// SIMATIC S7-200 SMART project (STEP 7-Micro/WIN SMART), CPU ST20

SYMBOL_TABLE 系统符号
Always_On        SM0.0    // 始终接通
First_Scan_On    SM0.1    // 仅在第一个扫描周期时接通
Clock_60s        SM0.4    // 针对 1 分钟的周期时间，时钟脉冲接通 30 s，断开 30 s.
Clock_1s         SM0.5    // 针对 1 s 的周期时间，时钟脉冲接通 0.5 s，断开 0.5 s.
END_SYMBOL_TABLE

ORGANIZATION_BLOCK MAIN:OB1
TITLE=// ============================================================
// // 文件: OB1_MAIN.stl
// // 功能: PLC主循环程序
// // 项目: 药液配置与加注控制系统
// // Story: AQEX-6 状态机骨架 + AQEX-9 急停调度顺序确认
// // PLC: S7-200 SMART CPU ST20
// // 说明: 本文件为语句表(STL)格式，可参考导入STEP 7-Micro/WIN SMART
// // 调度顺序: FC0(初始化)→FC2(急停,最高优先级)→FC4(Modbus)→FC3(报警)→FC22(RTC同步)
// //           →FC40(双倒计时器周期管理,v2.2新增)→FC1(状态调度)
// //           FC2在FC1之前,保证急停触发时同周期转S_ERROR
// //           FC40在FC1之前,保证M16.1下一轮S1触发脉冲及时响应
// //           【v2.2 修订 2026-09-15】FC40 从 FC1 内部调用移至 OB1 顶层调度
// // ============================================================
// 
// // 符号注释（实际导入时在符号表定义）
// // VW2     : 状态机当前状态 (0=S0,1=S1...8=S7,99=ERROR)
// // VW4     : 注射泵状态码
// // VW6     : 当前最高优先级报警码
// // VW8     : 实验总换水次数目标(=VD414×VD24/1440,单位:次)
// // V0.0    : CMD_Start (HMI→PLC启动命令)
// // V0.2    : CMD_Stop  (HMI→PLC停止命令)
// // V1.0    : STA_StartAck (PLC→HMI启动确认)
// // I1.1    : DI_EStop (急停反馈，常开NO，OFF=正常/ON=急停触发)  v1.3 改NO接法(原"常闭,ON=正常"注释已过期)
// // I0.3    : DI_Btn_SystemReset (系统复位按钮)
// 
BEGIN
Network 1
//  首次扫描初始化
//  SM0.1仅在首次扫描周期ON，调用FC0系统初始化
LD     First_Scan_On:SM0.1
=      L60.0                 // 局部存储器中转
LD     L60.0
CALL   SysInit:SBR0




// 急停与安全处理（每周期调用，优先级最高）
     // 急停与安全处理（每周期调用，优先级最高）
// SM0.0常ON，每周期调用FC2
        // SM0.0常ON，每周期调用FC2
LD     Always_On:SM0.0
CALL   EStopHandling:SBR2




// HMI停止命令(V0.2) - 自动运行中任意状态可停止
 // HMI停止命令(V0.2) - 自动运行中任意状态可停止
// ★ 2026-09-11 修复:
         // ★ 2026-09-11 修复:
//   (1) 去掉 AW< VW2, 99 条件,允许 S_ERROR 态(VW2=99)也能停止
 //   (1) 去掉 AW< VW2, 99 条件,允许 S_ERROR 态(VW2=99)也能停止
//       原逻辑只允许 VW2=1~8 停止, S_ERROR 锁死时点停止被忽略
 //       原逻辑只允许 VW2=1~8 停止, S_ERROR 锁死时点停止被忽略
//       新逻辑: VW2>0(非S0)就能停止, 急停/继电器故障锁存位由 FC19 管理
 //       新逻辑: VW2>0(非S0)就能停止, 急停/继电器故障锁存位由 FC19 管理
//   (2) 补清阀门诊断子状态 VB260~VB275 和诊断计时器 T50~T55
 //   (2) 补清阀门诊断子状态 VB260~VB275 和诊断计时器 T50~T55
//       原三个清理路径(停止/冷启动/复位)全部遗漏,导致
 //       原三个清理路径(停止/冷启动/复位)全部遗漏,导致
//       FC11/FC15/FC17 的 AW=VW2xx,0 前置条件不成立,
 //       FC11/FC15/FC17 的 AW=VW2xx,0 前置条件不成立,
//       开阀指令被跳过,表现为"点启动 M10.2=1 但系统不运行"
 //       开阀指令被跳过,表现为"点启动 M10.2=1 但系统不运行"
LD     V0.2
EU
AW>    VW2, 0                // VW2>0(排除S0), VW2=1~8 或 99 都允许停止
LPS
R      CPU_输出0:Q0.0, 7       // 泵停/阀关/NC电磁阀失电
R      T37, 1                // 停S1计时器
R      M10.2, 1              // 清S1首次进入标志
R      M10.7, 1              // 清预规划标志
R      M11.6, 1              // 清注射泵写请求
// ★ 新增: 清阀门诊断子状态+结果(VB260~VB275, 8字=16字节)
 // ★ 新增: 清阀门诊断子状态+结果(VB260~VB275, 8字=16字节)
//   覆盖: 阀A子状态VB260~261, 阀B子状态VB262~263,
 //   覆盖: 阀A子状态VB260~261, 阀B子状态VB262~263,
//         阀A/B结果VB266~269, 阀C诊断VB270~273, 其他辅助变量
 //         阀A/B结果VB266~269, 阀C诊断VB270~273, 其他辅助变量
FILL   0, VW260, 8
// ★ 新增: 清阀A/B诊断计时器 T50~T55
 // ★ 新增: 清阀A/B诊断计时器 T50~T55
R      T50, 6
// 【v2.2新增】停止时清理上缸子流程状态 + 双倒计时器标志 + 定时器
 // 【v2.2新增】停止时清理上缸子流程状态 + 双倒计时器标志 + 定时器
MOVW   0, VW418              // 上缸配液子流程状态清零
MOVW   0, VW400              // 换水计数清零 【v2.3.2迁移: 原VW306与手动命令位V306.0~V307.3重叠】
R      M16.0, 4              // M16.0~M16.3 连续清零
R      T38, 1                // 清 S2 搅拌定时器
R      T63, 1                // [已修复 v2.2] 清 1s 脉冲定时器
R      T49, 1                // 清 S4 转移计时器
MOVR   0.0, VD248            // [已修复 v2.2] 清 TimerA_Elapsed
MOVR   0.0, VD252            // [已修复 v2.2] 清 TimerB_Elapsed
MOVR   0.0, VD256            // 清 TimerA 显示值
MOVR   0.0, VD244            // 清 TimerB 显示值
MOVW   0, VW2                // 回S0
R      V0.2, 1               // 清停止命令
LPP




// Modbus通讯轮询（每周期调用）
        // Modbus通讯轮询（每周期调用）
LD     Always_On:SM0.0
CALL   ModbusPolling:SBR4




// 报警处理（每周期调用）
              // 报警处理（每周期调用）
LD     Always_On:SM0.0
CALL   AlarmHandling:SBR3




// RTC时间同步处理（每周期调用）
         // RTC时间同步处理（每周期调用）
// 处理HMI校时命令V0.6和5分钟超时保护
    // 处理HMI校时命令V0.6和5分钟超时保护
LD     Always_On:SM0.0
CALL   RTC_Sync:SBR24




// v2.2 双倒计时器周期管理（每周期调用）
    // v2.2 双倒计时器周期管理（每周期调用）
// ★ 必须在 FC1 状态调度之前调用,保证 M16.1 下一轮 S1 触发脉冲及时响应
 // ★ 必须在 FC1 状态调度之前调用,保证 M16.1 下一轮 S1 触发脉冲及时响应
// 替代原 AQEX-8 三层纠偏,严格保证 24h 换水次数硬约束 (VD414)
 // 替代原 AQEX-8 三层纠偏,严格保证 24h 换水次数硬约束 (VD414)
// 功能: 计算 T_cycle / 触发 S6 / 触发下一轮 S1 / 倒计时到 0 报警 / 双计时器显示值
 // 功能: 计算 T_cycle / 触发 S6 / 触发下一轮 S1 / 倒计时到 0 报警 / 双计时器显示值
LD     Always_On:SM0.0
CALL   RhythmCorrection:SBR19




// 【v2.3 新增】M16.1 唯一消费点: FC40 触发下一轮 S1 → 上缸 VW418 4→1
 // 【v2.3 新增】M16.1 唯一消费点: FC40 触发下一轮 S1 → 上缸 VW418 4→1
// 置位方只有 FC40 NET5 (Prep_Needed 且距周期末 ≥ T_prep), FC10/FC15 不再置位
 // 置位方只有 FC40 NET5 (Prep_Needed 且距周期末 ≥ T_prep), FC10/FC15 不再置位
// 【2026-09-29修复】同步置 M10.2(S1首次进入标志),与FC10首轮播种口径一致,
 // 【2026-09-29修复】同步置 M10.2(S1首次进入标志),与FC10首轮播种口径一致,
//   否则下一轮S1因FC11入口门(LD M10.2)不通而空转
 //   否则下一轮S1因FC11入口门(LD M10.2)不通而空转
LD     M16.1
MOVW   1, VW418
S      M10.2, 1
R      M16.1, 1




// 状态机调度(急停时FC2会强制VW2=99)
   // 状态机调度(急停时FC2会强制VW2=99)
// 每周期根据VW2调用对应状态FC
         // 每周期根据VW2调用对应状态FC
LD     Always_On:SM0.0
CALL   StateDispatcher:SBR1




// 【v2.2 新增】上缸子流程调度(VW418)
  // 【v2.2 新增】上缸子流程调度(VW418)
// 在 FC1 下缸调度之后调用,处理上缸 S1/S2 并行流程
 // 在 FC1 下缸调度之后调用,处理上缸 S1/S2 并行流程
// VW418=1 → CALL FC11_State_S1_Inlet (上缸进水)
 // VW418=1 → CALL FC11_State_S1_Inlet (上缸进水)
// VW418=2 → CALL FC1A_State_S2_MixDose (上缸搅拌+加药合并,v2.2 新建)
 // VW418=2 → CALL FC1A_State_S2_MixDose (上缸搅拌+加药合并,v2.2 新建)
// VW418=0/3/4 → 无动作(空闲/配完等待/已转移由其他 FC 处理)
 // VW418=0/3/4 → 无动作(空闲/配完等待/已转移由其他 FC 处理)
LD     Always_On:SM0.0
AW=    VW418, 1
AW>    VW2, 0                // 【2026-09-24修复】非S0(上缸随下缸运行才允许执行)
AW<    VW2, 99               // 【2026-09-24修复】非S_ERROR(故障锁定禁止上缸动作)
CALL   State_S1_Inlet:SBR6
LD     Always_On:SM0.0
AW=    VW418, 2
AW>    VW2, 0                // 【2026-09-24修复】同上
AW<    VW2, 99               // 【2026-09-24修复】同上
CALL   State_S2_MixDose:SBR7




// 手动控制处理（仅在S0态调用,在状态调度之后）
  // 手动控制处理（仅在S0态调用,在状态调度之后）
// 处理HMI画面3手动控制命令位V306.0~V307.1
 // 处理HMI画面3手动控制命令位V306.0~V307.1
//   (旧地址V2.4~V3.5因与VW2物理重叠已于2026-09-03迁移,详见FC20符号表)
 //   (旧地址V2.4~V3.5因与VW2物理重叠已于2026-09-03迁移,详见FC20符号表)
// 由FC20使用M13.0~M13.4锁存输出,NC电磁阀自动跟随(详见FC20)
 // 由FC20使用M13.0~M13.4锁存输出,NC电磁阀自动跟随(详见FC20)
LD     Always_On:SM0.0
LDW=   VW2, 0
CALL   ManualControl:SBR15




// 手动注射泵控制（仅在S0态调用,在手动阀门控制之后）
 // 手动注射泵控制（仅在S0态调用,在手动阀门控制之后）
// 处理V307.2/V307.3命令位
       // 处理V307.2/V307.3命令位
//   (旧地址V3.6/V3.7因与VW2物理重叠已于2026-09-03迁移,详见FC21符号表)
 //   (旧地址V3.6/V3.7因与VW2物理重叠已于2026-09-03迁移,详见FC21符号表)
// 【v2.5】由FC21壳使用VD452/VW388/VW390执行单次/循环抽排,
 // 【v2.5】由FC21壳使用VD452/VW388/VW390执行单次/循环抽排,
//   泵协议状态机与自动共用FC23引擎(详见FC21/FC23)
 //   泵协议状态机与自动共用FC23引擎(详见FC21/FC23)
LD     Always_On:SM0.0
LDW=   VW2, 0
CALL   ManualSyringePump:SBR23




// 非S0态清除手动控制锁存与手动注射泵状态,防止返回S0时误动作
 // 非S0态清除手动控制锁存与手动注射泵状态,防止返回S0时误动作
// 【v2.5】M13.5/M13.6保护标志已退役(FC23引擎取消),只清停止请求M13.7;
 // 【v2.5】M13.5/M13.6保护标志已退役(FC23引擎取消),只清停止请求M13.7;
//   追加手动模式残留子状态清除: 自动运行期间FC13壳已把M17.0刷0条件恒假,
 //   追加手动模式残留子状态清除: 自动运行期间FC13壳已把M17.0刷0条件恒假,
//   手动中途切自动时M17.0=1→清VW226,防引擎带旧子状态进入自动路径
 //   手动中途切自动时M17.0=1→清VW226,防引擎带旧子状态进入自动路径
LD     Always_On:SM0.0
LDW=   VW2, 0
NOT
R      M13.0, 5              // 清阀门/泵手动锁存
R      M13.7, 1              // 清停止请求(v2.5: M13.5/13.6已退役)
MOVW   0, VW390              // HMI状态镜像复位(空闲)
LDW=   VW2, 0
NOT
A      M17.0                 // 【v2.5】VW2≠0 且 手动模式残留
MOVW   0, VW226              // 清引擎子状态(FC23与FC13/FC21共用)
R      M17.0, 1




// M16.4/5/6 → V区镜像（供HMI读取，McgsPro S7-200 SMART以太网驱动不支持M区直接导入）
 // M16.4/5/6 → V区镜像（供HMI读取，McgsPro S7-200 SMART以太网驱动不支持M区直接导入）
// V1.1=InitDone(原M16.4), V1.2=RTU1/Syringe在线(原M16.5), V0.1=RTU2/Flow在线(原M16.6)
 // V1.1=InitDone(原M16.4), V1.2=RTU1/Syringe在线(原M16.5), V0.1=RTU2/Flow在线(原M16.6)
LD     Always_On:SM0.0
LD     M16.4
=      V1.1
LD     M16.5
=      V1.2
LD     M16.6
=      V0.1




// 系统总状态 → VB305 (0=良好,1=故障,2=急停)
 // 系统总状态 → VB305 (0=良好,1=故障,2=急停)
// 急停: I1.1=ON(NO触点,ON=急停触发) OR V300.4 OR V300.5
 // 急停: I1.1=ON(NO触点,ON=急停触发) OR V300.4 OR V300.5
// 故障: VW6≠0 AND 非急停
        // 故障: VW6≠0 AND 非急停
// 良好: 非急停 AND VW6=0 (默认值)
  // 良好: 非急停 AND VW6=0 (默认值)
// 【2026-09-24修复】v1.3改NO接法后此处漏改: 原"LD I1.1 / NOT"把I1.1=OFF(正常)误判为急停,
 // 【2026-09-24修复】v1.3改NO接法后此处漏改: 原"LD I1.1 / NOT"把I1.1=OFF(正常)误判为急停,
//   导致急停释放后HMI标题栏永久显示"急停"; 故障分支的"A I1.1"同步改为"AN I1.1"
 //   导致急停释放后HMI标题栏永久显示"急停"; 故障分支的"A I1.1"同步改为"AN I1.1"


LD     Always_On:SM0.0
MOVB   0, VB305              // 默认良好
// 急停 → 2
                   // 急停 → 2
LD     CPU_输入9:I1.1          // NO触点: ON=急停触发
O      V300.4
O      V300.5
MOVB   2, VB305
// 非急停 + 有报警 → 1
            // 非急停 + 有报警 → 1
LDW<>  VW6, 0
AN     CPU_输入9:I1.1          // 急停未触发(NO触点OFF=正常)
AN     V300.4
AN     V300.5
MOVB   1, VB305




// 实验总换水次数目标计算(v2.2新增)
      // 实验总换水次数目标计算(v2.2新增)
// VW8 = VD414(24h换水目标次数) × VD24(实验总时长min) / 1440
 // VW8 = VD414(24h换水目标次数) × VD24(实验总时长min) / 1440
// 供HMI画面显示实验全程应完成的总换水次数
    // 供HMI画面显示实验全程应完成的总换水次数
LD     Always_On:SM0.0
MOVR   VD414, AC0
*R     VD24, AC0
/R     1440.0, AC0
ROUND  AC0, AC0
DTI    AC0, VW8




// ============================================================
 // ============================================================
// 文件结束
                     // 文件结束
// 说明:
                      // 说明:
//   1. FC0/FC1/FC2/FC3/FC4 见各自独立文件
 //   1. FC0/FC1/FC2/FC3/FC4 见各自独立文件
//   2. FC10~FC19 各状态FC见 State_Sxx.stl 文件
 //   2. FC10~FC19 各状态FC见 State_Sxx.stl 文件
//   3. FC20 手动控制(新增,AQEX-34修复)
 //   3. FC20 手动控制(新增,AQEX-34修复)
//   4. FC22 RTC时间同步处理(新增,AQEX-51)
 //   4. FC22 RTC时间同步处理(新增,AQEX-51)
//   5. 导入时需先建符号表，再逐个新建FC并粘贴代码
 //   5. 导入时需先建符号表，再逐个新建FC并粘贴代码
//   6. VB305 系统状态字(=0良好/1故障/2急停,AQEX-50新增)
 //   6. VB305 系统状态字(=0良好/1故障/2急停,AQEX-50新增)
// ============================================================
 // ============================================================


END_ORGANIZATION_BLOCK

SUBROUTINE_BLOCK SysInit:SBR0
TITLE=// ============================================================
// // 文件: FC0_SysInit.stl (调度骨架)
// // 功能: 系统初始化入口 — 首次扫描 + Modbus清零 + 冷启/断电路径调度
// // Story: AQEX-6 + AQEX-11 + AQEX-51
// // 说明: 拆分自原单一 FC0,冷启/断电恢复逻辑分别独立到 SBR25/SBR26
// //   跨 SBR 无 JMP/LBL 依赖,每个 SBR 内部 LBL 空间独立
// // LBL 分配: FC0 用 1(断电恢复入口)、2(完成汇合)
// //          SBR25 用 8/9/10/88/89(冷启动)
// //          SBR26 用 1/3/4/5/6/7(断电恢复)
// //   跨 SBR 编号相同不冲突,POU 内 LBL 空间独立
// // 修复记录:
// //   2026-09-13: 拆分前 FC0 12KB 导致 STEP7 下载"块过大"误判,
// //               拆分后 FC0(~3KB) + SBR25(~4KB) + SBR26(~4KB) 三个小块
// // ============================================================
// 
// // 符号说明:
// // M16.4: M_InitDone        初始化完成标志(断电保持;v2.2迁移自V304.0,2026-09-15)
// // VW198 : VW_Init_Step      初始化步骤号(调试用,0=完成)
// // ColdStart  : SBR25 冷启动路径
// // WarmRecovery: SBR26 断电恢复路径
// 
// 
BEGIN
Network 1
//  SM0.1首次扫描 + Modbus库清零 + FC21计数器清零
//  ★ 2026-09-07修复: 每次首次扫描统一清零,库状态机在STOP→RUN后必须复位
LD     First_Scan_On:SM0.1
MOVW   1, VW198


LD     First_Scan_On:SM0.1
FILL   0, VW600, 143         // VB600~VB885清零(Modbus库存储区)
FILL   0, VW378, 2           // 清 VB378~VB381 (MBUS Error 4字节合并)
R      M10.0, 6              // 清M10.0~M10.5(Done位/降级标志)
R      M11.0, 1              // 清MBUS_CTRL Done位
MOVW   0, VW390              // 清手动注射泵子状态
R      M11.6, 1              // 清注射泵写请求
R      T104, 1               // 清回零冷却定时器




// 冷启/断电路径调度 + 完成汇合
         // 冷启/断电路径调度 + 完成汇合
// 判断冷启动/断电恢复
               // 判断冷启动/断电恢复
// M16.4=1 → JMP 1 (LBL 1: CALL WarmRecovery → JMP 2)
 // M16.4=1 → JMP 1 (LBL 1: CALL WarmRecovery → JMP 2)
// M16.4=0 → 冷启动 → CALL ColdStart → RET回 FC0 继续到 LBL 2
 // M16.4=0 → 冷启动 → CALL ColdStart → RET回 FC0 继续到 LBL 2
// 【v2.2迁移 2026-09-15】M_InitDone 从 V304.0 迁至 M16.4（位对象，无字节级冲突）
 // 【v2.2迁移 2026-09-15】M_InitDone 从 V304.0 迁至 M16.4（位对象，无字节级冲突）


LD     M16.4
JMP    1                     // M16.4=1 → 跳断电恢复路径


// ========== 冷启动路径 ==========
 // ========== 冷启动路径 ==========
LD     First_Scan_On:SM0.1
AN     M16.4                 // 冷启动(M16.4=0)
CALL   ColdStart:SBR25       // SBR25: 出厂硬编码 + 用户默认覆盖 + TODR + 安全初始化
                          // ColdStart 自然结束返回
 // ColdStart 自然结束返回
LD     Always_On:SM0.0
JMP    2                     // ★ 关键: 无条件跳过 LBL 1,否则会形成死循环


// ========== 断电恢复路径 ==========
 // ========== 断电恢复路径 ==========
LBL    1
LD     First_Scan_On:SM0.1
CALL   WarmRecovery:SBR26    // SBR26: TODR + RTC检测 + BCD转秒 + 状态机恢复
                          // WarmRecovery 自然结束后,顺序执行到 LBL 2 汇合
 // WarmRecovery 自然结束后,顺序执行到 LBL 2 汇合


// ========== 初始化完成汇合 ==========
 // ========== 初始化完成汇合 ==========
LBL    2
LD     First_Scan_On:SM0.1
S      M16.4, 1              // M_InitDone=1(初始化完成,断电保持;从V304.0迁移)
MOVW   0, VW198              // 步骤=0(完成)
// 汇合后自然结束 FC0,返回 OB1
       // 汇合后自然结束 FC0,返回 OB1




// ============================================================
 // ============================================================
// 文件结束
                     // 文件结束
// ============================================================
 // ============================================================


END_SUBROUTINE_BLOCK

SUBROUTINE_BLOCK StateDispatcher:SBR1
TITLE=// ============================================================
// // 文件: FC1_StateDispatcher.stl
// // 功能: 状态机调度器（每周期根据VW2调用对应下缸状态FC）
// // Story: v2.2 流程重构 (替代 AQEX-6 状态机骨架)
// // 说明: v2.2 取消上缸流程作为下缸主状态的 S1/S2/S3/S3.5
// //       上缸流程已拆出到 VW418 State_UpTank 子流程,由 OB1 NET 7 直接调度
// //       本 FC1 仅调度下缸 VW2 路径: S0/S4/S5/S6/S7/S_ERROR
// //   修复记录:
// //     P1-NETWORK标题去掉冒号(错误66)
// //     P2-JMP/LBL跨NETWORK问题修复: 全部合并到NETWORK 1
// //     【v2.2 修订 2026-09-15】删除 S1/S2/S3/S3.5 LBL;上缸流程外移至 OB1
// // ============================================================
BEGIN
Network 1
//  状态调度 (JMP/LBL必须在同一NETWORK内)
//  读取VW2并与各状态值比较，相等则调用对应FC
//  VW2 = 0 → S0初始化
JMP    1
// VW2 = 5 → S4上→下转移         // VW2 = 5 → S4上→下转移
LDW=   VW2, 5
JMP    2
// VW2 = 6 → S5实验运行中         // VW2 = 6 → S5实验运行中
LDW=   VW2, 6
JMP    3
// VW2 = 7 → S6下缸排水          // VW2 = 7 → S6下缸排水
LDW=   VW2, 7
JMP    4
// VW2 = 8 → S7实验结束          // VW2 = 8 → S7实验结束
LDW=   VW2, 8
JMP    5
// VW2 = 99 → S_ERROR故障锁定    // VW2 = 99 → S_ERROR故障锁定
LDW=   VW2, 99
JMP    6
// 其他非法值 → 强制回S0             // 其他非法值 → 强制回S0
LDW>=  VW2, 100
JMP    7
// 若未匹配任何状态(0<VW2<99但非上述值),也回S0 // 若未匹配任何状态(0<VW2<99但非上述值),也回S0
JMP    7
// S0入口                      // S0入口
LBL    1
CALL State_S0_Init
JMP    8
// S4入口                      // S4入口
LBL    2
CALL State_S4_Transfer
JMP    8
// S5入口                      // S5入口
LBL    3
CALL State_S5_Run
JMP    8
// S6入口                      // S6入口
LBL    4
CALL State_S6_Drain
JMP    8
// S7入口                      // S7入口
LBL    5
CALL State_S7_End
JMP    8
// S_ERROR入口                 // S_ERROR入口
LBL    6
CALL State_Error
JMP    8
// 非法状态处理(强制回S0)             // 非法状态处理(强制回S0)
LBL    7
LDW<=  VW2, 0                // VW2=0
// 调度结束                      // 调度结束
LBL    8
// 状态调度完成,返回 OB1             // 状态调度完成,返回 OB1
// 注: 上缸子流程(VW418=1/2)由 OB1 NET 7 在本 FC1 之后调度 // 注: 上缸子流程(VW418=1/2)由 OB1 NET 7 在本 FC1 之后调度
// ============================================================ // ============================================================
// 文件结束                      // 文件结束
// 说明:                       // 说明:
//   1. JMP/LBL必须在同一NETWORK内 //   1. JMP/LBL必须在同一NETWORK内
//   2. 每个状态FC内部负责状态转移(修改VW2) //   2. 每个状态FC内部负责状态转移(修改VW2)
//   3. 【v2.2】删除 S1/S2/S3/S3.5 入口:上缸流程移至 VW418 子流程 //   3. 【v2.2】删除 S1/S2/S3/S3.5 入口:上缸流程移至 VW418 子流程
//   4. 【v2.2】VW2 路径:0(S0)→5(S4)→6(S5)→7(S6)→8(S7) 或 99(S_ERROR) //   4. 【v2.2】VW2 路径:0(S0)→5(S4)→6(S5)→7(S6)→8(S7) 或 99(S_ERROR)
//   5. 【v2.2】VW418 路径:0(空闲)→1(S1)→2(S2搅拌+加药)→4(已转移) //   5. 【v2.2】VW418 路径:0(空闲)→1(S1)→2(S2搅拌+加药)→4(已转移)
//                          或 3(配完等待),由 OB1 NET 7 调度 FC11/FC1A //                          或 3(配完等待),由 OB1 NET 7 调度 FC11/FC1A
// ============================================================
 // ============================================================
JMP    1
LDW=   VW2, 5
JMP    2
LDW=   VW2, 6
JMP    3
LDW=   VW2, 7
JMP    4
LDW=   VW2, 8
JMP    5
LDW=   VW2, 99
JMP    6
LDW>=  VW2, 100
JMP    7
JMP    7
LBL    1
CALL   State_S0_Init:SBR5
JMP    8
LBL    2
CALL   State_S4_Transfer:SBR10
JMP    8
LBL    3
CALL   State_S5_Run:SBR11
JMP    8
LBL    4
CALL   State_S6_Drain:SBR12
JMP    8
LBL    5
CALL   State_S7_End:SBR13
JMP    8
LBL    6
CALL   State_Error:SBR14
JMP    8
LBL    7
MOVW   0, VW2
LBL    8
END_SUBROUTINE_BLOCK

SUBROUTINE_BLOCK EStopHandling:SBR2
TITLE=// ============================================================
// // 文件: FC2_EStopHandling.stl
// // 功能: 急停与安全处理（每周期调用，优先级最高）
// // Story: AQEX-6 状态机骨架 + AQEX-9 急停双通道+安全继电器反馈(详细实现)
// // 说明: 急停检测(I1.1 上升沿:NO 闭合)→锁存V300.4→转S_ERROR  v1.3 NO 进 I1.1
// //       安全继电器反馈延时校验(2秒)→V300.5继电器故障最高级报警
// //       输出强制安全(QB0=0,Q0.7声音开)
// //       急停解除与系统复位由FC19(State_Error)处理
// // ============================================================
// 
// // 符号说明:
// // I1.1  : DI_EStop           急停反馈(常开 NO,OFF=正常,ON=急停触发)  v1.3 改为接 NO 触点
// // I1.2  : DI_SafetyRelay_FB  安全继电器辅助反馈(ON=动力回路接通,OFF=动力回路断开)
// // V300.4: M_EStop_Latch      急停触发锁存(漫溢级,强制人工确认)
// // V300.5: M_Alarm_SafetyRelay 安全继电器故障(最高级,强制人工确认)
// // VW2   : 状态机状态(FC2写99转S_ERROR)
// // VW6   : 报警码(99=继电器故障,10=急停)
// // T35   : 安全继电器反馈延时(PT=20,2秒)
// // M10.7 : 预规划触发标志(急停时清,防止S5残留)
// 
// 
BEGIN
Network 1
//  急停触发+锁存+转S_ERROR + 安全继电器反馈校验 + 输出强制安全(合并NET 1-3)
//  [已修复 v2.2] 用 V62.6 缓存 EU 结果,避免 S/R 链栈空;删除直接写 VW6(由 FC3 根据 V300.x 计算)
LD     CPU_输入9:I1.1
EU
AN     First_Scan_On:SM0.1   // 首次扫描周期不触发（调试临时）
=      V62.6
LD     V62.6
S      V300.4, 1             // M_EStop_Latch锁存
LD     V62.6
MOVW   99, VW2               // VW2=99(转S_ERROR)
LD     V62.6
R      M10.7, 1              // 清预规划标志


// 安全继电器反馈延时校验(2秒内I1.2应OFF,否则继电器故障)
 // 安全继电器反馈延时校验(2秒内I1.2应OFF,否则继电器故障)
LD     V300.4
A      CPU_输入10:I1.2
TON    T35, 20
LD     T35
EU
S      V300.5, 1             // M_Alarm_SafetyRelay


// 急停锁存时输出强制安全
              // 急停锁存时输出强制安全
LD     V300.4
MOVB   0, QB0                // 泵停/阀关/NC电磁阀失电(安全)
S      CPU_输出7:Q0.7, 1       // 报警声音开




// 报警码写入(优先级:继电器故障99 > 急停10)
 // 报警码写入(优先级:继电器故障99 > 急停10)
// [已修复 v2.2] 删除直接写 VW6,统一由 FC3 NETWORK1 根据 V300.4/V300.5 计算
 // [已修复 v2.2] 删除直接写 VW6,统一由 FC3 NETWORK1 根据 V300.4/V300.5 计算
// LD     V300.5
            // LD     V300.5
// MOVW   99, VW6
           // MOVW   99, VW6
// LD     V300.4
            // LD     V300.4
// AN     V300.5
            // AN     V300.5
// MOVW   10, VW6
           // MOVW   10, VW6


LBL    1




// 注: HMI停止命令由OB1 MAIN NETWORK 3统一处理(VW2>0即可停止),本FC不再处理
 // 注: HMI停止命令由OB1 MAIN NETWORK 3统一处理(VW2>0即可停止),本FC不再处理
// 注: 急停解除与系统复位逻辑在FC19(State_Error)中处理
 // 注: 急停解除与系统复位逻辑在FC19(State_Error)中处理
// 注: Q8.0报警灯光由FC3 AlarmHandling按VW6优先级统一管理(Story 1.6)
 // 注: Q8.0报警灯光由FC3 AlarmHandling按VW6优先级统一管理(Story 1.6)
// 注: I1.2接线逻辑:ON=动力回路接通,OFF=动力回路断开(与代码注释一致)
 // 注: I1.2接线逻辑:ON=动力回路接通,OFF=动力回路断开(与代码注释一致)
// 注: 安全继电器反馈延时2秒兼顾机械动作时间与故障捕获灵敏度
 // 注: 安全继电器反馈延时2秒兼顾机械动作时间与故障捕获灵敏度
// 注: 急停硬件回路(安全继电器切断动力电)不经过PLC,本FC仅处理软件层面
 // 注: 急停硬件回路(安全继电器切断动力电)不经过PLC,本FC仅处理软件层面




// ============================================================
 // ============================================================
// 文件结束
                     // 文件结束
// ============================================================
 // ============================================================


END_SUBROUTINE_BLOCK

SUBROUTINE_BLOCK AlarmHandling:SBR3
TITLE=// ============================================================
// // 文件: FC3_AlarmHandling.stl
// // 功能: 报警处理（每周期调用）
// // Story: AQEX-6 状态机骨架 + AQEX-10 报警分级与消音/消光逻辑(详细实现)
// // 说明: 优先级链计算VW6 + 消音(I0.4/V0.4) + 消光(V0.3确认)
// //       自动恢复模式(V200.0=0时一般故障级条件消失自动复位)
// //       高优先级(漫溢/节奏滞后/继电器故障)强制人工确认,不受模式影响
// // ============================================================
// 
// // 符号说明:
// // VW6   : 当前最高优先级未确认报警码(0=无,99=继电器故障,10~14漫溢,20~21节奏,30~65一般)
// // V200.0: M_AlarmAckMode 报警确认模式(0=自动恢复,1=人工确认)
// // Q0.7  : 报警声音(FC2/FC19置位,FC3管理消音)
// // Q8.0  : 报警灯光(FC3统一管理,避免双写冲突)
// // I0.4  : 就地消音按钮(常开点动)
// // V0.3  : CMD_AckAlarm HMI报警确认命令
// // V0.4  : CMD_Mute HMI消音命令
// // V1.3  : STA_AlarmAckDone 报警确认握手
// // V1.4  : STA_MuteDone 消音握手
// // M11.1 : M_Sound_Latched 声音已消音标志(新报警时清,实现重鸣)
// // M11.2 : M_PrevAlarm 上一周期有报警标志(新报警检测用)
// 
// 
BEGIN
Network 1
//  优先级链计算 VW6(最高优先级未确认报警码)
//  压缩版: 用 LDW=+A+MOVW 条件赋值,替代 LD/JMP/LBL 结构
//  优先级: 99 > 10~14 > 20~21 > 66 > 30~36 > 40~47 > 49 > 60~61 > 64~65
//  【v10.4硬件变更】链中已移除: 13(V300.3)/45(V302.5)/47(V302.7)/61(V303.1),
//    对应位均改为保留位,当前有效码不含13/45/47/61
//  原理: 从最高优先级开始逐个检查,VW6一旦被赋值,后续 LDW= VW6,0 为假,自动跳过
LD     Always_On:SM0.0
MOVW   0, VW6                // 默认无报警


// 1. 安全继电器故障(99)
           // 1. 安全继电器故障(99)
LD     V300.5
MOVW   99, VW6


// 2. 漫溢级(10~14) - 逐位检查
     // 2. 漫溢级(10~14) - 逐位检查
// 【v10.4硬件变更】报警码13(V300.3,原NC球阀-下缸动作)已废弃,
 // 【v10.4硬件变更】报警码13(V300.3,原NC球阀-下缸动作)已废弃,
//   Q0.6去除后无任何FC置位V300.3,优先级链移除该条目(V300.3为保留位)
 //   Q0.6去除后无任何FC置位V300.3,优先级链移除该条目(V300.3为保留位)
LDW=   VW6, 0
A      V300.0
MOVW   10, VW6
LDW=   VW6, 0
A      V300.1
MOVW   11, VW6
LDW=   VW6, 0
A      V300.2
MOVW   12, VW6
LDW=   VW6, 0
A      V300.4
MOVW   14, VW6


// 3. 节奏滞后(20~21)
           // 3. 节奏滞后(20~21)
LDW=   VW6, 0
A      V300.6
MOVW   20, VW6
LDW=   VW6, 0
A      V300.7
MOVW   21, VW6


// 4. 单轮换水周期超时(66)
          // 4. 单轮换水周期超时(66)
LDW=   VW6, 0
A      V303.6
MOVW   66, VW6


// 5. 阀A类(30~36) - 逐位检查
     // 5. 阀A类(30~36) - 逐位检查
LDW=   VW6, 0
A      V301.0
MOVW   30, VW6
LDW=   VW6, 0
A      V301.2
MOVW   32, VW6
LDW=   VW6, 0
A      V301.3
MOVW   33, VW6
LDW=   VW6, 0
A      V301.4
MOVW   34, VW6
LDW=   VW6, 0
A      V301.5
MOVW   35, VW6
LDW=   VW6, 0
A      V301.6
MOVW   36, VW6


// 6. 阀B/C类(40~47) - 逐位检查
   // 6. 阀B/C类(40~47) - 逐位检查
// 【v10.4硬件变更】报警码45(V302.5)/47(V302.7)已废弃(I0.2去除,FC32不再置位),
 // 【v10.4硬件变更】报警码45(V302.5)/47(V302.7)已废弃(I0.2去除,FC32不再置位),
//   优先级链移除该两条目(V302.5/V302.7为保留位)
 //   优先级链移除该两条目(V302.5/V302.7为保留位)
LDW=   VW6, 0
A      V302.0
MOVW   40, VW6
LDW=   VW6, 0
A      V302.1
MOVW   41, VW6
LDW=   VW6, 0
A      V302.2
MOVW   42, VW6
LDW=   VW6, 0
A      V302.3
MOVW   43, VW6
LDW=   VW6, 0
A      V302.4
MOVW   44, VW6
LDW=   VW6, 0
A      V302.6
MOVW   46, VW6


// 7. 其他类(49,60,64,65)
      // 7. 其他类(49,60,64,65)
// 【v10.4硬件变更】报警码61(V303.1,原阀C关到位仍有流)已废弃(内漏判定依赖I0.2),
 // 【v10.4硬件变更】报警码61(V303.1,原阀C关到位仍有流)已废弃(内漏判定依赖I0.2),
//   优先级链移除该条目;报警码60(V303.0)现覆盖关到位超时+排水超时两种触发
 //   优先级链移除该条目;报警码60(V303.0)现覆盖关到位超时+排水超时两种触发
LDW=   VW6, 0
A      V303.2
MOVW   49, VW6
LDW=   VW6, 0
A      V303.0
MOVW   60, VW6
LDW=   VW6, 0
A      V303.4
MOVW   64, VW6
LDW=   VW6, 0
A      V303.5
MOVW   65, VW6




// 报警输出管理(灯光常亮 + 新报警声音重鸣)
   // 报警输出管理(灯光常亮 + 新报警声音重鸣)
// 有活动报警(VW6≠0) → 灯光Q8.0常亮
  // 有活动报警(VW6≠0) → 灯光Q8.0常亮
// 新报警(VW6由0变非0) → 清M_Sound_Latched,声音重鸣
 // 新报警(VW6由0变非0) → 清M_Sound_Latched,声音重鸣
LDW<>  VW6, 0
S      EM0_输出0:Q8.0, 1       // 灯光常亮


// 新报警检测: 本周期VW6≠0 且 上一周期M11.2=0(无报警) → 新报警
 // 新报警检测: 本周期VW6≠0 且 上一周期M11.2=0(无报警) → 新报警
LDW<>  VW6, 0
AN     M11.2                 // 上一周期无报警 → 新报警
R      M11.1, 1              // 清消音标志(新报警重鸣)


// 声音管理: 有报警且未消音 → 声音开
      // 声音管理: 有报警且未消音 → 声音开
LDW<>  VW6, 0
AN     M11.1                 // 未消音
S      CPU_输出7:Q0.7, 1       // 声音开


// 自动恢复模式: VW6=0且自动模式 → 自动消光
 // 自动恢复模式: VW6=0且自动模式 → 自动消光
LDW=   VW6, 0
AN     V200.0                // M_AlarmAckMode=0(自动模式)
R      EM0_输出0:Q8.0, 1       // 无报警自动消光
R      CPU_输出7:Q0.7, 1       // 无报警关声音
R      M11.1, 1              // 清消音标志


// 更新上一周期报警标志
               // 更新上一周期报警标志
LDW<>  VW6, 0
=      M11.2                 // 记录本周期有报警(供下周期新报警检测)




// 消音处理(I0.4就地按钮 OR V0.4 HMI命令)
 // 消音处理(I0.4就地按钮 OR V0.4 HMI命令)
// [已修复 v2.2] 用 V62.7 缓存消音请求,避免 OLD 后 S/R 链栈空
 // [已修复 v2.2] 用 V62.7 缓存消音请求,避免 OLD 后 S/R 链栈空
// 消音源: I0.4上升沿 OR V0.4上升沿
  // 消音源: I0.4上升沿 OR V0.4上升沿
LD     CPU_输入4:I0.4
EU
LD     V0.4
EU
OLD                          // 两者任一上升沿
=      V62.7
LD     V62.7
R      CPU_输出7:Q0.7, 1       // 关声音
LD     V62.7
S      M11.1, 1              // 置消音标志(新报警时清)
LD     V62.7
S      V1.4, 1               // STA_MuteDone握手
LD     V62.7
R      V0.4, 1               // 清HMI消音命令
// 注: 消音只关声音,灯光Q8.0和报警位保持;新报警(VW6变化)时M11.1清,声音重鸣
 // 注: 消音只关声音,灯光Q8.0和报警位保持;新报警(VW6变化)时M11.1清,声音重鸣




// 报警确认处理(V0.3 HMI确认 → 条件消失才消光+清锁存)
 // 报警确认处理(V0.3 HMI确认 → 条件消失才消光+清锁存)
// V0.3上升沿 = HMI报警确认命令(高优先级HMI侧二次确认,PLC只收V0.3)
 // V0.3上升沿 = HMI报警确认命令(高优先级HMI侧二次确认,PLC只收V0.3)
// 确认规则: V0.3上升沿后,逐个检查报警位条件,条件消失的复位报警位,再由NETWORK1重算VW6
 // 确认规则: V0.3上升沿后,逐个检查报警位条件,条件消失的复位报警位,再由NETWORK1重算VW6
// ★ 关键修复(2026-09-04): NETWORK 4 缺 V0.3 上升沿门控(JMP),导致每周期无条件
 // ★ 关键修复(2026-09-04): NETWORK 4 缺 V0.3 上升沿门控(JMP),导致每周期无条件
//   执行所有条件复位,包括 LD V303.5; R V303.5, 1——使 S_ERROR 立即被清
 //   执行所有条件复位,包括 LD V303.5; R V303.5, 1——使 S_ERROR 立即被清
//   修复: V0.3 无上升沿时跳过整个网络,避免误清报警位
 //   修复: V0.3 无上升沿时跳过整个网络,避免误清报警位
// ★★★ 2026-09-11 发现 JMP 条件写反了！ ★★★
 // ★★★ 2026-09-11 发现 JMP 条件写反了！ ★★★
//   原代码 LD V0.3; EU; JMP 40：EU=1(有上升沿)时跳转 → 反而跳过了 R V0.3,1
 //   原代码 LD V0.3; EU; JMP 40：EU=1(有上升沿)时跳转 → 反而跳过了 R V0.3,1
//   正确：用 V60.5 缓存 EU 结果,LDN 取反后触发 JMP,再用 LD 恢复栈顶执行线圈
 //   正确：用 V60.5 缓存 EU 结果,LDN 取反后触发 JMP,再用 LD 恢复栈顶执行线圈
//   注意：STL 的 S/R/= 线圈指令依赖栈顶=1 才执行,不能用 NOT+JMP（会清掉栈顶）
 //   注意：STL 的 S/R/= 线圈指令依赖栈顶=1 才执行,不能用 NOT+JMP（会清掉栈顶）
//   注意：S7-200 SMART 不支持 JMPN 指令,必须用 JMP + LDN 中转
 //   注意：S7-200 SMART 不支持 JMPN 指令,必须用 JMP + LDN 中转
LD     V0.3
EU
=      V60.5                 // 缓存 EU 结果: 有上升沿=1, 无上升沿=0
LDN    V60.5                 // 无上升沿时栈顶=1
JMP    40                    // ★ 无上升沿则跳转到 LBL 40,跳过确认处理
LD     V60.5                 // 有上升沿时栈顶=1,恢复执行条件


S      V1.3, 1               // STA_AlarmAckDone握手
R      V0.3, 1               // 清确认命令


// 漫溢级: 条件消失才复位(液位计高位=OFF)
  // 漫溢级: 条件消失才复位(液位计高位=OFF)
LD     V300.0                // 上缸漫溢
AN     CPU_输入5:I0.5          // 液位计A-高位已OFF
R      V300.0, 1             // 复位
LD     V300.1                // 下缸漫溢
AN     CPU_输入7:I0.7          // 液位计B-高位已OFF
R      V300.1, 1
// NC阀动作: 由人工确认复位(无DI直接条件,保持锁存需HMI强制,此处不自动复位)
 // NC阀动作: 由人工确认复位(无DI直接条件,保持锁存需HMI强制,此处不自动复位)
// 急停V300.4/继电器故障V300.5: 由FC19系统复位按钮/HMI高权限确认处理,FC3不碰
 // 急停V300.4/继电器故障V300.5: 由FC19系统复位按钮/HMI高权限确认处理,FC3不碰


// 节奏滞后级: 条件消失(新一轮开始)由FC40重置,FC3不直接处理
 // 节奏滞后级: 条件消失(新一轮开始)由FC40重置,FC3不直接处理
// 但V0.3确认时,若V300.6/7已由FC40清除,NETWORK1会重算VW6
 // 但V0.3确认时,若V300.6/7已由FC40清除,NETWORK1会重算VW6


// 一般故障级: 条件消失则复位(调用公共子程序,与 NETWORK 5 共享)
 // 一般故障级: 条件消失则复位(调用公共子程序,与 NETWORK 5 共享)
CALL   AlarmReset_Common:SBR28


// 单轮换水周期超时(66): V0.3人工确认复位 + 双计时器清零(本轮重新计时)
 // 单轮换水周期超时(66): V0.3人工确认复位 + 双计时器清零(本轮重新计时)
// 【2026-09-25补漏】V303.6置位后原无任何复位路径(锁存到冷启动);
 // 【2026-09-25补漏】V303.6置位后原无任何复位路径(锁存到冷启动);
//   FC40设计注4要求此报警"不受V200.0模式影响,必须V0.3人工确认",
 //   FC40设计注4要求此报警"不受V200.0模式影响,必须V0.3人工确认",
//   故不放FC3A(避免NETWORK 5自动模式复用),仅在V0.3上升沿(本网络已门控)复位;
 //   故不放FC3A(避免NETWORK 5自动模式复用),仅在V0.3上升沿(本网络已门控)复位;
//   必须同时清零VD248/VD252: OB1中FC3先于FC40执行,若只清报警位,
 //   必须同时清零VD248/VD252: OB1中FC3先于FC40执行,若只清报警位,
//   NET6同扫描会因"Elapsed仍>=T_cycle且NET4被VW6=66封锁"立即重报形成死锁;
 //   NET6同扫描会因"Elapsed仍>=T_cycle且NET4被VW6=66封锁"立即重报形成死锁;
//   清零后条件消失,下一扫描VW6=0解锁NET4,节奏自动恢复
 //   清零后条件消失,下一扫描VW6=0解锁NET4,节奏自动恢复
LD     Always_On:SM0.0
R      V303.6, 1
MOVR   0.0, VD248            // 确认=本轮重新计时
MOVR   0.0, VD252


LBL    40                    // ★ NETWORK 4 跳转目标(无V0.3上升沿时跳过确认处理)


// 注: 报警位复位后,下一周期NETWORK1重算VW6;若VW6=0,NETWORK2自动消光
 // 注: 报警位复位后,下一周期NETWORK1重算VW6;若VW6=0,NETWORK2自动消光
// 注: 漫溢级(V300.0~2;V300.3已废弃为保留位)、急停(V300.4)、继电器故障(V300.5)不由FC3复位
 // 注: 漫溢级(V300.0~2;V300.3已废弃为保留位)、急停(V300.4)、继电器故障(V300.5)不由FC3复位
//      由FC19系统复位按钮/HMI高权限确认处理
 //      由FC19系统复位按钮/HMI高权限确认处理




// 自动恢复模式(M_AlarmAckMode=0时一般故障级条件消失自动复位)
 // 自动恢复模式(M_AlarmAckMode=0时一般故障级条件消失自动复位)
// 自动模式: V200.0=0时,一般故障级报警位条件消失自动R复位
 // 自动模式: V200.0=0时,一般故障级报警位条件消失自动R复位
// 漫溢/节奏滞后/继电器故障不受此模式影响,保持锁存
 // 漫溢/节奏滞后/继电器故障不受此模式影响,保持锁存
// ★ 2026-09-11 修复 AQEX-XX: 状态机已进S_ERROR(VW2=99)时禁止自动清报警位
 // ★ 2026-09-11 修复 AQEX-XX: 状态机已进S_ERROR(VW2=99)时禁止自动清报警位
//   原因: 一般故障触发MOVW 99,VW2后，若自动恢复立即清报警位，
 //   原因: 一般故障触发MOVW 99,VW2后，若自动恢复立即清报警位，
//   会导致 VW2=99 + VW6=0 的状态机/报警系统不一致
 //   会导致 VW2=99 + VW6=0 的状态机/报警系统不一致
//   场景: 阀A开到位超时(V301.4)后阀A终于开到位(I8.0=ON),
 //   场景: 阀A开到位超时(V301.4)后阀A终于开到位(I8.0=ON),
//         FC3 NETWORK 5 自动清V301.4→VW6=0,但VW2已锁99无人解锁,
 //         FC3 NETWORK 5 自动清V301.4→VW6=0,但VW2已锁99无人解锁,
//         OB1 NETWORK12 按VW6=0算VB305=0(良好),掩盖故障
 //         OB1 NETWORK12 按VW6=0算VB305=0(良好),掩盖故障
//   防御: S_ERROR态暂停自动恢复,让FC19 NETWORK5自动解锁或人工复位处理
 //   防御: S_ERROR态暂停自动恢复,让FC19 NETWORK5自动解锁或人工复位处理
LDW=   VW2, 99
JMP    50                    // S_ERROR态 → 跳过自动恢复,报警位保持


LD     V200.0                // M_AlarmAckMode
NOT                          // =0(自动模式)时执行后续


// 一般故障级: 条件消失则复位(调用公共子程序,与 NETWORK 4 共享)
 // 一般故障级: 条件消失则复位(调用公共子程序,与 NETWORK 4 共享)
CALL   AlarmReset_Common:SBR28


LBL    50                    // ★ S_ERROR态跳过自动恢复的跳转目标(2026-09-11新增)


// 注: 漫溢(V300.0~3)、急停(V300.4)、继电器故障(V300.5)、节奏滞后(V300.6/7)不在此处理
 // 注: 漫溢(V300.0~3)、急停(V300.4)、继电器故障(V300.5)、节奏滞后(V300.6/7)不在此处理
// 注: V303.6(单轮换水周期超时)也不在自动恢复范围,必须由V0.3人工确认(FC3 NETWORK 4)
 // 注: V303.6(单轮换水周期超时)也不在自动恢复范围,必须由V0.3人工确认(FC3 NETWORK 4)
// 注: 自动复位后下一周期NETWORK1重算VW6,NETWORK2自动消光
 // 注: 自动复位后下一周期NETWORK1重算VW6,NETWORK2自动消光




// NETWORK 6 报警日志已删除(压缩体积)
  // NETWORK 6 报警日志已删除(压缩体积)
// HMI 侧已有完整报警历史记录,PLC 仅保留 VW6 供 HMI 轮询即可
 // HMI 侧已有完整报警历史记录,PLC 仅保留 VW6 供 HMI 轮询即可




// ============================================================
 // ============================================================
// 文件结束
                     // 文件结束
// 说明:
                      // 说明:
//   1. FC3每周期调用,负责报警码计算+输出管理+确认处理+自动恢复+日志
 //   1. FC3每周期调用,负责报警码计算+输出管理+确认处理+自动恢复+日志
//   2. 报警位置位由各FC(FC2/FC30~32/FC40等)负责,FC3只复位
 //   2. 报警位置位由各FC(FC2/FC30~32/FC40等)负责,FC3只复位
//   3. Q8.0灯光由FC3统一管理,FC2/FC19不操作Q8.0(避免双写)
 //   3. Q8.0灯光由FC3统一管理,FC2/FC19不操作Q8.0(避免双写)
//   4. Q0.7声音由FC2/FC19置位(急停/故障态),FC3管理消音+新报警重鸣
 //   4. Q0.7声音由FC2/FC19置位(急停/故障态),FC3管理消音+新报警重鸣
//   5. 编址修正: M_AlarmAckMode=V200.0(避VD124冲突),SafetyRelayAck=V0.7(避V0.5冲突)
 //   5. 编址修正: M_AlarmAckMode=V200.0(避VD124冲突),SafetyRelayAck=V0.7(避V0.5冲突)
//   6. 高优先级(漫溢/节奏滞后/继电器故障)强制人工确认,不受M_AlarmAckMode影响
 //   6. 高优先级(漫溢/节奏滞后/继电器故障)强制人工确认,不受M_AlarmAckMode影响
//   7. NETWORK4/5的报警位复位条件需与各FC置位条件严格对应(现场调试时核实)
 //   7. NETWORK4/5的报警位复位条件需与各FC置位条件严格对应(现场调试时核实)
// ============================================================
 // ============================================================


END_SUBROUTINE_BLOCK

SUBROUTINE_BLOCK ModbusPolling:SBR4
TITLE=
BEGIN
Network 1
//    MBUS_CTRL: 9600/8/N/1, 超时1000ms
LD     Always_On:SM0.0
=      L60.0
LD     Always_On:SM0.0
=      L63.7
LD     L60.0
CALL   MBUS_CTRL:SBR20, L63.7, 9600, 16#0, 16#0, 1000, M11.0, VB378
//   T103: MBUS_MSG超时定时器(100ms时基, PT=100=10s)
 //   T103: MBUS_MSG超时定时器(100ms时基, PT=100=10s)
//   任一任务活跃(M15.0~M15.4)时计时, 超时后强制切换任务
 //   任一任务活跃(M15.0~M15.4)时计时, 超时后强制切换任务
LD     M15.0
O      M15.1
O      M15.2
O      M15.3
O      M15.4
TON    T103, 100
//   任务0: 注射泵状态读(41001)
     //   任务0: 注射泵状态读(41001)
//   EN=VW290==0 AND M15.0, First=M15.0上升沿(EU)
 //   EN=VW290==0 AND M15.0, First=M15.0上升沿(EU)
LDW=   VW290, 0
=      L60.0
LD     M15.0
EU
=      L63.7
LD     L60.0
CALL   MBUS_MSG:SBR21, L63.7, 16#1, 16#0, 16#A029, 16#1, &VB410, M10.0, VB379
//   任务1: 流量计读(40009)
       //   任务1: 流量计读(40009)
//   EN=VW290==1 AND M15.1, First=M15.1上升沿(EU)
 //   EN=VW290==1 AND M15.1, First=M15.1上升沿(EU)
LDW=   VW290, 1
=      L60.0
LD     M15.1
EU
=      L63.7
LD     L60.0
CALL   MBUS_MSG:SBR21, L63.7, 16#2, 16#0, 16#9C49, 16#2, &VB410, M14.0, VB380
//   任务2: 注射泵位置读(41007)
     //   任务2: 注射泵位置读(41007)
//   EN=VW290==2 AND M15.2, First=M15.2上升沿(EU)
 //   EN=VW290==2 AND M15.2, First=M15.2上升沿(EU)
LDW=   VW290, 2
=      L60.0
LD     M15.2
EU
=      L63.7
LD     L60.0
CALL   MBUS_MSG:SBR21, L63.7, 16#1, 16#0, 16#A02F, 16#1, &VB410, M10.1, VB381
//   任务3: 流量计瞬时流量读(40007) → VD94
 //   任务3: 流量计瞬时流量读(40007) → VD94
//   EN=VW290==3 AND M15.3, First=M15.3上升沿(EU)
 //   EN=VW290==3 AND M15.3, First=M15.3上升沿(EU)
LDW=   VW290, 3
=      L60.0
LD     M15.3
EU
=      L63.7
LD     L60.0
CALL   MBUS_MSG:SBR21, L63.7, 16#2, 16#0, 16#9C47, 16#2, &VB410, M14.1, VB382
//   === 任务0: 成功/失败/切换 合并 (原 7/12/13) ===
 //   === 任务0: 成功/失败/切换 合并 (原 7/12/13) ===
//   任务0成功处理: VW410->VW224(原始状态码暂存), 成功计数, 清失败计数
 //   任务0成功处理: VW410->VW224(原始状态码暂存), 成功计数, 清失败计数
//   【2026-10-08修复 v2.3.9】原"直接MOVW VW410, VW4"导致VW4=原始码(96/64/100),
 //   【2026-10-08修复 v2.3.9】原"直接MOVW VW410, VW4"导致VW4=原始码(96/64/100),
//   而FC13/FC3A全部按归一化值(0就绪/1空闲/2运动中)判断:
 //   而FC13/FC3A全部按归一化值(0就绪/1空闲/2运动中)判断:
//   FC13子状态1写命令门控AW= VW4,0恒假→加药指令永不下发,VW226卡子状态1
 //   FC13子状态1写命令门控AW= VW4,0恒假→加药指令永不下发,VW226卡子状态1
//   →S2不加药不退出。现恢复"原始码暂存VW224+下方归一化NETWORK"两级结构。
 //   →S2不加药不退出。现恢复"原始码暂存VW224+下方归一化NETWORK"两级结构。
LD     M10.0
A      M15.0
AB=    VB379, 0
MOVW   VW410, VW224
AENO
MOVW   0, VW292
AENO
R      V303.4, 1
//   【2026-09-29修复】置位注射泵RTU在线标志: v2.2迁移丢失置位点(与M10.2同族)
 //   【2026-09-29修复】置位注射泵RTU在线标志: v2.2迁移丢失置位点(与M10.2同族)
//   只在此块(读成功)置位, 连续失败达滤波阈值(5次)才离线(见下方)
 //   只在此块(读成功)置位, 连续失败达滤波阈值(5次)才离线(见下方)
S      M16.5, 1
//   任务0失败计数
                //   任务0失败计数
LD     M10.0
A      M15.0
AB<>   VB379, 0
INCW   VW292
//   【2026-09-29修复】注射泵连续读失败≥5次 → 离线标志复位
 //   【2026-09-29修复】注射泵连续读失败≥5次 → 离线标志复位
LDW>=  VW292, 5
R      M16.5, 1
//   任务0完成切换(成功或T103超时)
     //   任务0完成切换(成功或T103超时)
//   [已修复 v2.2] 用 V60.1 保存切换条件，避免 LD+O+R 后栈空导致后续指令失效
 //   [已修复 v2.2] 用 V60.1 保存切换条件，避免 LD+O+R 后栈空导致后续指令失效
LD     M10.0
O      T103
=      V60.1
LD     V60.1
R      M15.0, 1
LD     V60.1
S      M15.1, 1
LD     V60.1
MOVW   1, VW290
LD     V60.1
R      M10.0, 1
LD     V60.1
R      T103, 1
//   [已修复 v2.2] 删除 VW224→VW4 归一化死代码。任务0成功时已直接 MOVW VW410, VW4。
 //   [已修复 v2.2] 删除 VW224→VW4 归一化死代码。任务0成功时已直接 MOVW VW410, VW4。
//   ★2026-10-08撤销上述删除(v2.3.9): 经FC99现场确认泵原始码为96/64/100/103,
 //   ★2026-10-08撤销上述删除(v2.3.9): 经FC99现场确认泵原始码为96/64/100/103,
//   直接搬运使FC13加药门控AW= VW4,0恒假,加药死锁。归一化代码为必需而非死代码。
 //   直接搬运使FC13加药门控AW= VW4,0恒假,加药死锁。归一化代码为必需而非死代码。
//   === 任务0: VW4归一化 (原始码→0/1/2/4, 供FC13/FC3A使用) ===
 //   === 任务0: VW4归一化 (原始码→0/1/2/4, 供FC13/FC3A使用) ===
//   96(就绪/激活)→0, 64(空闲/休眠)→1, 97(初始化,上电自检瞬态)→1(v2.5.1,
 //   96(就绪/激活)→0, 64(空闲/休眠)→1, 97(初始化,上电自检瞬态)→1(v2.5.1,
//   原归4会把自检期设备误报成错误触发急停), 100(运动中)→2,
 //   原归4会把自检期设备误报成错误触发急停), 100(运动中)→2,
//   其他(含103未初始化/65~111错误码)→4(错误)
 //   其他(含103未初始化/65~111错误码)→4(错误)
//   结构: 先默认4(错误), 已知码依次覆盖——比4分支互斥比较节省程序体积
 //   结构: 先默认4(错误), 已知码依次覆盖——比4分支互斥比较节省程序体积
//   (2026-10-08 v2.3.9: ST20程序存储器12KB,警告830超界,压缩指令数)
 //   (2026-10-08 v2.3.9: ST20程序存储器12KB,警告830超界,压缩指令数)
LD     Always_On:SM0.0
MOVW   4, VW4                // 默认=错误
LDW=   VW224, 96
MOVW   0, VW4
LDW=   VW224, 64
MOVW   1, VW4
LDW=   VW224, 97
MOVW   1, VW4                // 【v2.5.1】初始化瞬态按空闲处理
LDW=   VW224, 100
MOVW   2, VW4
//   === 任务1: 成功/失败/切换 合并 (原 14/15/16) ===
 //   === 任务1: 成功/失败/切换 合并 (原 14/15/16) ===
//   任务1成功处理: VD410->VD86, 成功计数, 清失败计数
 //   任务1成功处理: VD410->VD86, 成功计数, 清失败计数
//   流量计32位浮点数据已按正确顺序存储,直接搬运即可
 //   流量计32位浮点数据已按正确顺序存储,直接搬运即可
LD     M14.0
A      M15.1
AB=    VB380, 0
MOVD   VD410, VD86
AENO
MOVW   0, VW294
//   【2026-09-29修复】置位流量计RTU在线标志: v2.2迁移丢失置位点(与M10.2同族)
 //   【2026-09-29修复】置位流量计RTU在线标志: v2.2迁移丢失置位点(与M10.2同族)
//   只在此块(读成功)置位, 连续失败达滤波阈值(5次)才离线(见下方)
 //   只在此块(读成功)置位, 连续失败达滤波阈值(5次)才离线(见下方)
S      M16.6, 1
//   【2026-09-24修复】删除"AENO / R V303.6"：V303.6 已于 2026-09-08 起划归 FC40
 //   【2026-09-24修复】删除"AENO / R V303.6"：V303.6 已于 2026-09-08 起划归 FC40
//   报警66(单轮换水周期超时)，此处残留复位会在流量计读成功时悄悄清掉周期超时报警
 //   报警66(单轮换水周期超时)，此处残留复位会在流量计读成功时悄悄清掉周期超时报警
//   任务1失败计数
                //   任务1失败计数
LD     M14.0
A      M15.1
AB<>   VB380, 0
INCW   VW294
//   【2026-09-29修复】流量计连续读失败≥5次 → 离线标志复位
 //   【2026-09-29修复】流量计连续读失败≥5次 → 离线标志复位
LDW>=  VW294, 5
R      M16.6, 1
//   任务1完成切换(成功或T103超时)
     //   任务1完成切换(成功或T103超时)
//   [已修复 v2.2] 用 V60.2 保存切换条件，避免 LD+O+R 后栈空导致后续指令失效
 //   [已修复 v2.2] 用 V60.2 保存切换条件，避免 LD+O+R 后栈空导致后续指令失效
LD     M14.0
O      T103
=      V60.2
LD     V60.2
R      M15.1, 1
LD     V60.2
S      M15.2, 1
LD     V60.2
MOVW   2, VW290
LD     V60.2
R      M14.0, 1
LD     V60.2
R      T103, 1
//   === 任务2: 成功/失败/切换 合并 (原 17/18/19) ===
 //   === 任务2: 成功/失败/切换 合并 (原 17/18/19) ===
//   任务2成功处理: VW410->VW222, 成功计数, 清失败计数
 //   任务2成功处理: VW410->VW222, 成功计数, 清失败计数
LD     M10.1
A      M15.2
AB=    VB381, 0
MOVW   VW410, VW222
AENO
MOVW   0, VW296
//   任务2失败计数
                //   任务2失败计数
LD     M10.1
A      M15.2
AB<>   VB381, 0
INCW   VW296
//   任务2完成切换(成功或T103超时)
     //   任务2完成切换(成功或T103超时)
//   [已修复 v2.2] 用 V60.6 保存切换条件，避免 LD+O+R 后栈空导致后续指令失效
 //   [已修复 v2.2] 用 V60.6 保存切换条件，避免 LD+O+R 后栈空导致后续指令失效
LD     M10.1
O      T103
=      V60.6
LD     V60.6
R      M15.2, 1
LD     V60.6
S      M15.3, 1
LD     V60.6
MOVW   3, VW290
LD     V60.6
R      M10.1, 1
LD     V60.6
R      T103, 1
//   === 任务3: 成功/失败/切换 合并 (原 20/21/22-25) ===
 //   === 任务3: 成功/失败/切换 合并 (原 20/21/22-25) ===
//   任务3成功处理: VD410->VD94(瞬时流量), 成功计数, 清失败计数
 //   任务3成功处理: VD410->VD94(瞬时流量), 成功计数, 清失败计数
//   流量计32位浮点数据已按正确顺序存储,直接搬运即可
 //   流量计32位浮点数据已按正确顺序存储,直接搬运即可
LD     M14.1
A      M15.3
AB=    VB382, 0
MOVD   VD410, VD94
AENO
MOVW   0, VW298
//   任务3失败计数
                //   任务3失败计数
LD     M14.1
A      M15.3
AB<>   VB382, 0
INCW   VW298
//   任务3完成切换: 有写请求 → 任务4, 否则 → 任务0
 //   任务3完成切换: 有写请求 → 任务4, 否则 → 任务0
//   用V60.0做完成事件中间继电器(仅此处赋值,无冲突)
 //   用V60.0做完成事件中间继电器(仅此处赋值,无冲突)
LD     M14.1
O      T103
=      V60.0
//  // 复位任务3相关标志
            //  // 复位任务3相关标志
LD     V60.0
R      M15.3, 1
R      M14.1, 1
R      T103, 1
//  // 进入任务4: 有写请求(M11.6=1)
 //  // 进入任务4: 有写请求(M11.6=1)
LD     V60.0
A      M11.6
S      M15.4, 1
MOVW   4, VW290
//  // 未进入任务4则回任务0
          //  // 未进入任务4则回任务0
LD     V60.0
AN     M15.4
S      M15.0, 1
MOVW   0, VW290
//   === 任务4: 写数据准备 + 写命令 合并 (原 27/29/30) ===
 //   === 任务4: 写数据准备 + 写命令 合并 (原 27/29/30) ===
//   任务4写数据准备: 有写请求时把VW230复制到统一缓冲区VW410
 //   任务4写数据准备: 有写请求时把VW230复制到统一缓冲区VW410
//   DataPtr用&VB410, 避免直接使用&VW230导致MBUS_MSG写失败(Error=104)
 //   DataPtr用&VB410, 避免直接使用&VW230导致MBUS_MSG写失败(Error=104)
LD     M11.6
MOVW   VW230, VW410
//   任务4: 注射泵写命令(仅在M11.6=1时执行)
 //   任务4: 注射泵写命令(仅在M11.6=1时执行)
//   EN=VW290==4 AND M15.4 AND M11.6, First=M15.4上升沿(EU)
 //   EN=VW290==4 AND M15.4 AND M11.6, First=M15.4上升沿(EU)
//   写目标地址VD232由FC0/FC13/FC21设置(16#9C42=40002强停,16#9C43=40003复位,16#9C46=40006抽液,16#9C47=40007排液)
 //   写目标地址VD232由FC0/FC13/FC21设置(16#9C42=40002强停,16#9C43=40003复位,16#9C46=40006抽液,16#9C47=40007排液)
LDW=   VW290, 4
A      M15.4
A      M11.6
=      V60.3
LDW=   VW290, 4
A      M15.4
A      M11.6
=      L60.0
LD     M15.4
EU
=      L63.7
LD     L60.0
CALL   MBUS_MSG:SBR21, L63.7, 16#1, 16#1, VD232, 16#1, &VB410, M12.0, VB383
//   === 任务4: 成功/失败/切换 合并 (原 31/32/33) ===
 //   === 任务4: 成功/失败/切换 合并 (原 31/32/33) ===
//   任务4成功处理: 清写请求, 成功计数, 清失败计数
 //   任务4成功处理: 清写请求, 成功计数, 清失败计数
//   ★关键: 写完成后立即清M11.6, 防止复位命令在轮询中反复写
 //   ★关键: 写完成后立即清M11.6, 防止复位命令在轮询中反复写
LD     M12.0
A      M15.4
AB=    VB383, 0
R      M11.6, 1
R      M11.7, 1
MOVW   0, VW510
R      V303.4, 1
//   任务4失败计数 + 从站异常立即报警
     //   任务4失败计数 + 从站异常立即报警
LD     M12.0
A      M15.4
LPS
AB<>   VB383, 0
INCW   VW510
LPP
AB>=   VB383, 101
S      V303.4, 1
//   任务4完成切换(成功或T103超时)
     //   任务4完成切换(成功或T103超时)
//   [已修复 v2.2] 用 V60.7 保存切换条件，避免 LD+O+R 后栈空导致后续指令失效
 //   [已修复 v2.2] 用 V60.7 保存切换条件，避免 LD+O+R 后栈空导致后续指令失效
//   R M15.4, S M15.0, 更新VW290=0, 清握手, 清超时定时器
 //   R M15.4, S M15.0, 更新VW290=0, 清握手, 清超时定时器
//  // ★M12.0不清! 由FC13/FC21请求方清零, 否则请求方看不到写完成
 //  // ★M12.0不清! 由FC13/FC21请求方清零, 否则请求方看不到写完成
LD     M12.0
O      T103
=      V60.7
LD     V60.7
R      M11.6, 1
LD     V60.7
R      M11.7, 1
LD     V60.7
R      M15.4, 1
LD     V60.7
S      M15.0, 1
LD     V60.7
MOVW   0, VW290
LD     V60.7
R      T103, 1
//   === 软件滤波 合并 (原 34/35/36) ===
 //   === 软件滤波 合并 (原 34/35/36) ===
//   V303.4软件滤波: 连续读失败<5次时不报警
 //   V303.4软件滤波: 连续读失败<5次时不报警
LDW<   VW292, 5
R      V303.4, 1
//   V303.4写任务软件滤波: 连续写失败<5次且无从站异常时不报警
 //   V303.4写任务软件滤波: 连续写失败<5次且无从站异常时不报警
LDW<   VW510, 5
AB<    VB383, 101
R      V303.4, 1
//   【2026-09-24修复】删除 V303.6 软件滤波(VW294<5 时复位)：V303.6 已划归 FC40
 //   【2026-09-24修复】删除 V303.6 软件滤波(VW294<5 时复位)：V303.6 已划归 FC40
//   报警66(单轮换水周期超时)，Modbus任务1失败不再使用此位(通讯失败报警待Story1.1)
 //   报警66(单轮换水周期超时)，Modbus任务1失败不再使用此位(通讯失败报警待Story1.1)




END_SUBROUTINE_BLOCK

SUBROUTINE_BLOCK State_S0_Init:SBR5
TITLE=// ============================================================
// // 文件: FC10_State_S0_Init.stl
// // 功能: S0初始化状态 (VW2=0)
// // Story: v2.2 流程重构 (替代 AQEX-6 状态机骨架)
// // 说明: v2.2 首轮由 FC10 一次性触发上缸 S1 (VW418=1) + 下缸进 S5 空等
// //       后续轮次由 FC17 在 S6 完成时切 M16.0 并清 M16.1,触发下一轮 S1
// //   修复记录:
// //     2026-09-11 新增硬件液位开关检查 (I0.6)
// //     【v2.2 修订 2026-09-15】首轮触发上缸 VW418=1 + 下缸 VW2=6 (S5 空等)
// //     【2026-09-29修复】启动网络重写: 补M10.2置位(v2.2丢失,致阀A永不动作) + V0.0两条路径都消费
// // ============================================================
BEGIN
Network 1
//  S0状态输出(安全待命)
//  仅复位Q0.0~Q0.6(泵/阀/NC电磁阀),Q0.7报警声音由FC3统一管理
//  【v10.4硬件变更】Q0.6(下缸NC阀)已去除,保留未使用;R Q0.0,7清零无害
LD     Always_On:SM0.0
R      CPU_输出0:Q0.0, 7       // 泵停、阀A/B/C关、上缸NC阀失电,保留Q0.7




// v2.2 首轮启动逻辑
              // v2.2 首轮启动逻辑
// 启动条件:
                    // 启动条件:
//   V0.0↑(CMD_Start 上升沿)
   //   V0.0↑(CMD_Start 上升沿)
//   AND VW6=0  (无活动报警)
     //   AND VW6=0  (无活动报警)
//   AND I0.6=ON (上缸排空,NPN常闭,液体低于探针闭合)
 //   AND I0.6=ON (上缸排空,NPN常闭,液体低于探针闭合)
// 启动动作(一次性播种):
             // 启动动作(一次性播种):
//   1. VW418 = 1 (上缸直接进入 S1 进水, OB1 上缸调度 FC11;
 //   1. VW418 = 1 (上缸直接进入 S1 进水, OB1 上缸调度 FC11;
//      首轮不再需要 M16.1 触发脉冲, 避免与 FC40 NET5 触发路径双写)
 //      首轮不再需要 M16.1 触发脉冲, 避免与 FC40 NET5 触发路径双写)
//   2. S M10.2 = 1 (S1首次进入标志) 【2026-09-29修复】v2.2重构丢失的置位点:
 //   2. S M10.2 = 1 (S1首次进入标志) 【2026-09-29修复】v2.2重构丢失的置位点:
//      无此置位则FC11入口门(LD M10.2/AW=VW260,0)永不通,阀A/上缸NC阀/诊断全部不启动
 //      无此置位则FC11入口门(LD M10.2/AW=VW260,0)永不通,阀A/上缸NC阀/诊断全部不启动
//   3. 清 M16.1 (防御性清旧触发脉冲, 首轮不置位)
 //   3. 清 M16.1 (防御性清旧触发脉冲, 首轮不置位)
//   4. S M16.0 = 1 (首轮固定使用 TimerA)
 //   4. S M16.0 = 1 (首轮固定使用 TimerA)
//   5. MOVW 6, VW2 (下缸直接进 S5 空等,不经过 S1/S2/S3/S4)
 //   5. MOVW 6, VW2 (下缸直接进 S5 空等,不经过 S1/S2/S3/S4)
//   6. S V1.0 (启动确认)
       //   6. S V1.0 (启动确认)
//   7. R V0.0 (清启动命令位,成功/失败两条路径都消费)
 //   7. R V0.0 (清启动命令位,成功/失败两条路径都消费)


// 【2026-09-29修复】原LPS/LPP+NOT+双LBL结构存在两个隐患:
 // 【2026-09-29修复】原LPS/LPP+NOT+双LBL结构存在两个隐患:
//   (a) M10.2无置位点(本次修复);
   //   (a) M10.2无置位点(本次修复);
//   (b) 条件不满足(JMP 1)时V0.0不被消费,启动命令悬空至HMI松键,语义不干净;
 //   (b) 条件不满足(JMP 1)时V0.0不被消费,启动命令悬空至HMI松键,语义不干净;
//   改为V60.0/V60.1草稿位缓存(与FC11的V61.1同套路),去掉全部栈操作。
 //   改为V60.0/V60.1草稿位缓存(与FC11的V61.1同套路),去掉全部栈操作。
// 注意: V60.0/V60.1为FC10专用扫描周期内草稿位,不跨块、不保持。
 // 注意: V60.0/V60.1为FC10专用扫描周期内草稿位,不跨块、不保持。


// 缓存启动脉冲(本扫描周期内有效)
         // 缓存启动脉冲(本扫描周期内有效)
LD     V0.0
EU
=      V60.0


// 三个条件全满足 → 允许播种
           // 三个条件全满足 → 允许播种
LD     V60.0
AW=    VW6, 0
A      CPU_输入6:I0.6
=      V60.1


// v2.2 首轮启动(一次性播种)
         // v2.2 首轮启动(一次性播种)
LD     V60.1
MOVW   1, VW418              // 【v2.3修复】首轮直接播种上缸 S1 (原清0无意义,首轮无入口则液体永远转不下去)
S      M10.2, 1              // 【2026-09-29修复】补S1首次进入标志置位(FC11入口门)
R      M16.1, 1              // 防御性清旧触发脉冲(后续轮次由 OB1 消费 M16.1 置 VW418=1)
S      M16.0, 1              // 首轮固定使用 TimerA (VD248)
// 【v2.2】下缸直接进 S5 空等(S4 转移由 FC40/FC17 触发,不再由 VW2=1~4 推进)
 // 【v2.2】下缸直接进 S5 空等(S4 转移由 FC40/FC17 触发,不再由 VW2=1~4 推进)
MOVW   6, VW2                // VW2=6 (S5 实验运行态,S5 等待 S4 转移条件)
S      V1.0, 1               // STA_StartAck=1


// 消费启动命令(仅脉冲周期执行;成功/失败两条路径都清,避免命令悬空)
 // 消费启动命令(仅脉冲周期执行;成功/失败两条路径都清,避免命令悬空)
LD     V60.0
R      V0.0, 1




// 注: 急停触发由 FC2 强制 VW2=99,此处不处理
 // 注: 急停触发由 FC2 强制 VW2=99,此处不处理
// 注: S7 实验结束后 HMI 确认重启也走此路径(经 S_ERROR 解除后回 S0)
 // 注: S7 实验结束后 HMI 确认重启也走此路径(经 S_ERROR 解除后回 S0)
// 注: v2.2 与 v2.1 关键区别: 首轮不再走 S1→S2→S3→S4 串行上电逻辑
 // 注: v2.2 与 v2.1 关键区别: 首轮不再走 S1→S2→S3→S4 串行上电逻辑
//       上缸配液 (VW418 子流程) 与下缸实验 (VW2 路径) 并行
 //       上缸配液 (VW418 子流程) 与下缸实验 (VW2 路径) 并行


// ============================================================
 // ============================================================
// 文件结束
                     // 文件结束
// ============================================================
 // ============================================================


END_SUBROUTINE_BLOCK

SUBROUTINE_BLOCK State_S1_Inlet:SBR6
TITLE=// ============================================================
// // 文件: FC11_State_S1_Inlet.stl
// // 功能: S1上缸进水 (VW2=1)
// // Story: AQEX-6 状态机骨架 + AQEX-7 阀门诊断(已集成) + AQEX-8 节奏纠偏(已集成二次校正)
// // 说明: 开阀A进水，调用FC30阀A诊断(差值法+延时验证)
// //       诊断结果VW266: 0进行中/1正常完成/2故障
// //       诊断正常完成 → 调用FC40二次校正(模式1) → 更新VD_T_Rolling → 转S2
// // ============================================================
// 
// // 符号说明:
// // VW260 : Diag_State_A  阀A诊断子状态
// // VW266 : Diag_Result_A 阀A诊断结果
// // VW278 : VD_Timeout_ValveA×10 转换值(供FC30的T50用,已修正避FC32冲突)
// // VW280 : VD_Delay_ValveA_Verify×10 转换值(供FC30的T51用)
// // VD332 : VD358运算中间变量(避免修改HMI参数VD358)
// // VD316 : 目标进水量(HMI设定,SBR25冷启动默认10L,用户默认区VD500覆盖)
// 
// 
BEGIN
Network 1
//  S1首次进入 - 开阀A+NC球阀+复位+流量计快照+参数计算+启动诊断(合并)
//  [已修复 v2.2] 用 V61.1 缓存 M10.2 AND VW260=0 条件,避免 S/R 指令链栈空
LD     M10.2
AW=    VW260, 0
=      V61.1
LD     V61.1
S      CPU_输出2:Q0.2, 1       // 开阀A
LD     V61.1
S      CPU_输出5:Q0.5, 1       // 开上缸NC球阀
LD     V61.1
R      T37, 1                // 复位S1计时器
LD     V61.1
R      T51, 1                // ★修复2026-09-30: 防御性清T51残留done位(子状态5报警路径不复位T51)
LD     Always_On:SM0.0
TON    T37, 32767            // 【v2.3.6修复2026-09-30】输入改SM0.0: 原V61.1单扫描脉冲致T37永不计时,VD70恒0                  // 【v2.3修复】启动S1实测计时(原只复位不启动,导致VD70恒为0)
LD     V61.1
R      V1.6, 1               // 置上缸状态=空
LD     V61.1
MOVD   VD86, VD82            // 流量计快照
LD     V61.1
MOVR   VD358, VD332          // 计算超时参数 VW278
*R     10.0, VD332
ROUND  VD332, AC0
MOVW   AC0, VW278
LD     V61.1
MOVR   VD66, VD320           // 计算延时参数 VW280
*R     10.0, VD320
ROUND  VD320, AC0
MOVW   AC0, VW280
LD     V61.1
MOVW   1, VW260
MOVB   0, VB266              // 清诊断结果
MOVB   0, VB267




// v2.3 双倒计时器: S1 首次进入时清零【非活动】Elapsed 计数器
 // v2.3 双倒计时器: S1 首次进入时清零【非活动】Elapsed 计数器
// 【v2.3修复】原"清零当前活动计数器"与流水线时序矛盾:
 // 【v2.3修复】原"清零当前活动计数器"与流水线时序矛盾:
//   S1 由 FC40 按"本轮剩余<=Prep_Needed"触发,启动于本轮中段,
 //   S1 由 FC40 按"本轮剩余<=Prep_Needed"触发,启动于本轮中段,
//   活动计数器正服务本轮(NET4/NET6节奏判定),清零会导致本轮节奏失效;
 //   活动计数器正服务本轮(NET4/NET6节奏判定),清零会导致本轮节奏失效;
//   非活动计数器属于下一轮,其计时从本轮S6完成切换后才开始,此处清零安全。
 //   非活动计数器属于下一轮,其计时从本轮S6完成切换后才开始,此处清零安全。
LDW=   VW418, 1              // 上缸进入 S1
AN     M16.2                 // S1 尚未开始(防止重复启动)
S      M16.2, 1              // 置 S1 已开始标志
LD     M16.0                 // 当前活动计时器为 TimerA?
MOVR   0.0, VD252            // 清零【非活动】TimerB_Elapsed
LDN    M16.0                 // 当前活动计时器为 TimerB?
MOVR   0.0, VD248            // 清零【非活动】TimerA_Elapsed




// 调用阀A诊断FC30
               // 调用阀A诊断FC30
LD     Always_On:SM0.0
CALL   ValveA_Diag:SBR16




// 检查阀A诊断结果 + 二次校正 + 转S2
    // 检查阀A诊断结果 + 二次校正 + 转S2
// ★ 关键: FC30 用 MOVB 写 VB266(只写低字节,高字节VB267=0)
 // ★ 关键: FC30 用 MOVB 写 VB266(只写低字节,高字节VB267=0)
//   所以 VW266 = VB266×256, 必须用 LDB= 字节比较,不能用 AW= 字比较
 //   所以 VW266 = VB266×256, 必须用 LDB= 字节比较,不能用 AW= 字比较
//   字节值 0=进行中, 1=正常完成, 2=故障(FC30已转S_ERROR)
 //   字节值 0=进行中, 1=正常完成, 2=故障(FC30已转S_ERROR)
LDB=   VB266, 1              // 诊断正常完成(字节比较,与FC30的MOVB匹配)
JMP    1                     // 是 → 跳转处理
LD     Always_On:SM0.0
JMP    2                     // 否 → 结束本NETWORK


LBL    1
LD     Always_On:SM0.0
MOVW   T37, VW236            // 【v2.3修复】先读当前值再复位(R在前读到的恒为0)
ITD    VW236, VD444          // 整数→双整数
DTR    VD444, VD70
/R     10.0, VD70            // 【v2.3.6】100ms时基→秒                  // 双整数→实数(VD_S1_Actual)
R      T37, 1                // 停S1计时(读后复位)
// 【v2.2 修订 2026-09-15】删除原 Story1.4 二次校正 FC40 调用
 // 【v2.2 修订 2026-09-15】删除原 Story1.4 二次校正 FC40 调用
// v2.2 取消三层纠偏,FC40 改为双倒计时器周期管理(由 OB1 顶层调用)
 // v2.2 取消三层纠偏,FC40 改为双倒计时器周期管理(由 OB1 顶层调用)
// 原 VD354/VW182/VW184/VD150/154/158 全部废弃
 // 原 VD354/VW182/VW184/VD150/154/158 全部废弃
// 保留位置仅为保留 S1 完成 → 转 S2/VW418=2 的状态机逻辑
 // 保留位置仅为保留 S1 完成 → 转 S2/VW418=2 的状态机逻辑


// 【v2.2 新增】S1 完成时清 M16.2 (S1 已开始标志) + 切 M16.0 (计时器切换, 由 FC17 S6 完成时切)
 // 【v2.2 新增】S1 完成时清 M16.2 (S1 已开始标志) + 切 M16.0 (计时器切换, 由 FC17 S6 完成时切)
LD     Always_On:SM0.0
R      M16.2, 1              // 清 S1 已开始标志
R      M16.3, 1              // 清 S2 首次进入标志(防御性)


// 【v2.2】S1 完成 → 转 VW418=2 (上缸 S2 搅拌+加药)
 // 【v2.2】S1 完成 → 转 VW418=2 (上缸 S2 搅拌+加药)
// v2.2 取消原"二次校正 VW184≠4"条件,改为无条件转移
 // v2.2 取消原"二次校正 VW184≠4"条件,改为无条件转移
// (FC40 已删除三层纠偏, 不再有"人工介入→S_ERROR"分支)
 // (FC40 已删除三层纠偏, 不再有"人工介入→S_ERROR"分支)
// 累加本次进水量到本次实验累计流量
         // 累加本次进水量到本次实验累计流量
MOVR   VD90, AC0             // AC0 = VD_Current_InletVolume
+R     AC0, VD406            // VD_ExpTotal_Flow += 本次进水量 (原VD364,2026-09-29迁移:与VD366重叠2字节;VD402槽被VW402(T38_PT)占)
MOVW   2, VW418              // 状态转移 S1→S2 (v2.2: VW418 上缸子流程而非 VW2)
R      M10.2, 1              // 清S1首次进入标志
R      T38, 1                // 进入S2前复位T38(防御性,FC1A 首次进入会再次启动 T38)


LBL    2




// 注: 漫溢保护、差值法计量、延时验证、内漏检测、开关到位诊断
 // 注: 漫溢保护、差值法计量、延时验证、内漏检测、开关到位诊断
//      全部由FC30统一处理，FC11仅负责状态转移调度
 //      全部由FC30统一处理，FC11仅负责状态转移调度
// 注: VD316(目标进水量)由HMI设定或SBR25用户默认覆盖写入,FC30用它做达标比较
 // 注: VD316(目标进水量)由HMI设定或SBR25用户默认覆盖写入,FC30用它做达标比较
// 注: 二次校正(Story 1.4)在转S2前调用
 // 注: 二次校正(Story 1.4)在转S2前调用
// 注: VD358运算已改用独立中间变量VD332,不再修改HMI设定参数
 // 注: VD358运算已改用独立中间变量VD332,不再修改HMI设定参数
// 注: 断电恢复由FC0统一处理,VW2=1(S1阀A动作中断)时FC0转S_ERROR
 // 注: 断电恢复由FC0统一处理,VW2=1(S1阀A动作中断)时FC0转S_ERROR




// ============================================================
 // ============================================================
// 文件结束
                     // 文件结束
// ============================================================
 // ============================================================


END_SUBROUTINE_BLOCK

SUBROUTINE_BLOCK State_S2_MixDose:SBR7
TITLE=// ============================================================
// // 文件: FC1A_State_S2_MixDose.stl
// // 功能: S2 搅拌 + 加药合并子状态 (VW418=2)
// // Story: v2.2 流程重构 - 新建(由原 FC12 + FC13 合并)
// // 说明: v2.2 取消独立 S3 加药子状态,改为"搅拌 + 加药"组合子状态
// //       潜水泵常开(整个 S2 期间不停),T38 计时到达 VD28 (固定搅拌时长) + VW226=9 (加药完成)
// //       共同触发 VW418=3 (上缸配完等待转移)
// //       【2026-10-08 v2.3.9】T38改SM0.0驱动,修复单扫描脉冲致永不计时
// //
// // 调用方: OB1 NET 7 仅在 VW418=2 时调用本 FC
// // 关联 FC: 本 FC 内部调用 FC13(自动壳) → CALL FC23_PumpEngine 完成加药
// //         子状态机逻辑(v2.5引擎化; VW226 0~9 语义不变,仅由本 FC 触发)
// //
// // 【v2.2 合并说明】
// //   - 原 FC12(预循环搅拌)功能: S2 启动潜水泵 + T38 计时 → 已集成到本 FC NETWORK 1
// //   - 原 FC13(加药)功能: VW226 0~9 子状态机(15 个 NETWORK) → 本 FC 内部 CALL FC13
// //   - 原 FC14(S3.5 静止等候)功能: 取消(v2.2 取消静止等候环节)
// // ============================================================
// // 符号说明:
// // VW402 : T38_PT  S2搅拌定时器PT(VD28×10, v2.3.2由VW252迁入,避让VD252 TimerB_Elapsed低字)
// // VW226 : 加药子状态机 (0~9, FC13内部使用)
// 
BEGIN
Network 1
//  首次进入 S2 - 启动潜水泵 + T38 计时 + 初始化加药子状态机
//  触发条件: VW418=2 (上缸 S2 入口) + M16.3=0 (首次进入门控)
//  启动动作: 开潜水泵1/2 + T38 PT = VD28 × 10 + 清 VW226 + R 注射泵异常 + 初始化 VD372/VD440
//  [已修复 v2.2] 用 V61.2 缓存 S2 首次进入条件,避免 S/R/LPS 后栈空
LDW=   VW418, 2
AN     M16.3
=      V61.2
LD     V61.2
S      M16.3, 1              // 置 S2 首次进入标志
LD     V61.2
S      CPU_输出0:Q0.0, 1       // 潜水泵1开
LD     V61.2
S      CPU_输出1:Q0.1, 1       // 潜水泵2开
LD     V61.2
MOVR   VD28, VD336           // T38 PT = VD28 × 10
*R     10.0, VD336
ROUND  VD336, AC0
MOVW   AC0, VW402            // VW402 = T38 PT 【v2.3.2迁移: 原VW252与VD252(TimerB_Elapsed REAL)低字重叠,互踩】
// 【2026-10-08修复 v2.3.9】T38输入改SM0.0: 原V61.2为首次进入单扫描脉冲,
 // 【2026-10-08修复 v2.3.9】T38输入改SM0.0: 原V61.2为首次进入单扫描脉冲,
//   TON输入断开即复位,搅拌定时器永不累计,T38永不到点→S2完成判定
 //   TON输入断开即复位,搅拌定时器永不累计,T38永不到点→S2完成判定
//   (VW226=9 AND T38)永不成立,S2无限滞留。与v2.3.6修T37同款。
 //   (VW226=9 AND T38)永不成立,S2无限滞留。与v2.3.6修T37同款。
//   安全性: FC1A仅被OB1在VW418=2时调用,SM0.0驱动等价于"S2期间持续计时";
 //   安全性: FC1A仅被OB1在VW418=2时调用,SM0.0驱动等价于"S2期间持续计时";
//   转出S2后FC1A不再被调用,T38停止刷新,完成/停止/复位路径均有R T38兜底。
 //   转出S2后FC1A不再被调用,T38停止刷新,完成/停止/复位路径均有R T38兜底。
LD     Always_On:SM0.0
TON    T38, VW402            // 启动 S2 搅拌定时器(S2全程计时)
LD     V61.2
MOVW   0, VW226              // 清 VW226 加药子状态机
LD     V61.2
R      V303.4, 1             // 清注射泵异常报警
LD     V61.2
MOVR   VD584, VD372          // VD_Remaining_Vol = 目标加药量
LD     V61.2
MOVR   0.0, VD440            // 累计加药量清零




// 调用 FC13(自动壳) → FC23 注射泵引擎完成加药子状态机(v2.5引擎化)
 // 调用 FC13(自动壳) → FC23 注射泵引擎完成加药子状态机(v2.5引擎化)
// FC23 内部使用 VW226 子状态推进加药流程(自动路径):
 // FC23 内部使用 VW226 子状态推进加药流程(自动路径):
//   0: 初始化(VD372=VD584)   1: 写抽液   2: 等抽液运动   3: 强停1
 //   0: 初始化(VD372=VD584)   1: 写抽液   2: 等抽液运动   3: 强停1
//   4: 等就绪1   5: 写排液   6: 等排液运动   7: 强停2   8: 结算/循环
 //   4: 等就绪1   5: 写排液   6: 等排液运动   7: 强停2   8: 结算/循环
//   9: 完成闩锁(本FC消费)   手动专用30/40/99见FC23文件头
 //   9: 完成闩锁(本FC消费)   手动专用30/40/99见FC23文件头
LD     Always_On:SM0.0
CALL   State_S3_Dosing:SBR8




// 完成判定 - 搅拌计时到 AND 加药子状态 9 → VW418=3 (上缸配完等待转移)
 // 完成判定 - 搅拌计时到 AND 加药子状态 9 → VW418=3 (上缸配完等待转移)
// [已修复 v2.2] 用 V61.3 缓存完成条件,避免 R 指令链栈空
 // [已修复 v2.2] 用 V61.3 缓存完成条件,避免 R 指令链栈空
// 潜水泵在判定完成后停止(Q0.0/Q0.1 复位)
 // 潜水泵在判定完成后停止(Q0.0/Q0.1 复位)
LDW=   VW226, 9              // 加药子状态 9 = 已完成
A      T38                   // 搅拌 T38 计时到
=      V61.3
LD     V61.3
R      CPU_输出0:Q0.0, 1       // 潜水泵1关
LD     V61.3
R      CPU_输出1:Q0.1, 1       // 潜水泵2关
LD     V61.3
R      T38, 1                // 清 T38
LD     V61.3
MOVW   3, VW418              // 上缸进入"配完等待转移"




// 注: S2 期间潜水泵与加药并行(同时进行),而非原"先搅拌后加药"
 // 注: S2 期间潜水泵与加药并行(同时进行),而非原"先搅拌后加药"
// 注: T38 计时由 VD28 (S2 固定时长) 决定,v2.2 严格不可压缩
 // 注: T38 计时由 VD28 (S2 固定时长) 决定,v2.2 严格不可压缩
// 注: VW226=9 + T38 到达 共同触发 VW418=3 (任一未达都不转)
 // 注: VW226=9 + T38 到达 共同触发 VW418=3 (任一未达都不转)
// 注: 故障时 FC13 内部已置 V303.4 并转 S_ERROR,由 FC19 处理
 // 注: 故障时 FC13 内部已置 V303.4 并转 S_ERROR,由 FC19 处理
// 注: 断电恢复时 VW418=2 由 SBR26 决定是否保持(详见 SBR26)
 // 注: 断电恢复时 VW418=2 由 SBR26 决定是否保持(详见 SBR26)


// ============================================================
 // ============================================================
// 文件结束
                     // 文件结束
// ============================================================
 // ============================================================


END_SUBROUTINE_BLOCK

SUBROUTINE_BLOCK State_S3_Dosing:SBR8
TITLE=// ============================================================
// // 文件: FC13_State_S3_Dosing.stl
// // 功能: 自动加药壳(v2.5) — 模式置自动+搅拌泵断言,泵协议见FC23引擎
// // 项目: 药液配置与加注控制系统
// // Story: v2.5 注射泵引擎化合并 — 本文件由"完整加药状态机"瘦身为"自动壳"
// // PLC: S7-200 SMART CPU ST20
// // 说明: 本文件为语句表(STL)格式，可参考导入STEP 7-Micro/WIN SMART
// //
// // 【2026-10-08 v2.5】原FC13的VW226子状态机(0~9)整体迁入FC23_PumpEngine,
// //   自动/手动共用。本壳保留自动路径的工艺职责:
// //     1. 模式位M17.0=0(引擎错误分流/完成分支依据,每扫描刷新)
// //     2. 搅拌泵Q0.0/Q0.1断言(完整生命周期归FC1A: S2入口S/完成R,
// //        此处同原FC13 NET1作进入时再断言)
// //     3. CALL PumpEngine
// //   引擎行为与本文件v2.4.0版逐NETWORK等价(状态0~9平移,全局错误门控
// //   由"VW418=2"改为"VW226≠0且≠99",在仅VW418=2调用的上下文下等价)。
// //
// // 调用方: FC1A_State_S2_MixDose (VW418=2时CALL State_S3_Dosing)
// // 完成语义: 引擎VW226=9闩锁, FC1A判"9 AND T38"→VW418=3, 与v2.2~v2.4一致
// // ============================================================
// 
BEGIN
Network 1
//  模式=自动(引擎错误→CALL PumpErrExit转S_ERROR; 完成→9闩锁)
LD     Always_On:SM0.0
R      M17.0, 1


// 搅拌泵断言(原FC13 NET1: 进入加药时开泵; FC1A握有S2全程生命周期)
 // 搅拌泵断言(原FC13 NET1: 进入加药时开泵; FC1A握有S2全程生命周期)
LD     Always_On:SM0.0
AW=    VW226, 0
S      CPU_输出0:Q0.0, 1       // 潜水泵1开
S      CPU_输出1:Q0.1, 1       // 潜水泵2开


// 调用注射泵引擎(协议状态机见FC23_PumpEngine.stl)
 // 调用注射泵引擎(协议状态机见FC23_PumpEngine.stl)
LD     Always_On:SM0.0
CALL   PumpEngine:SBR9




// ============================================================
 // ============================================================
// 文件结束
                     // 文件结束
// 说明:
                      // 说明:
//   1. 本壳不含任何泵协议逻辑,修改泵行为请改FC23(自动手动同时生效)
 //   1. 本壳不含任何泵协议逻辑,修改泵行为请改FC23(自动手动同时生效)
//   2. 自动目标VD584/剩余VD372/累计VD440由引擎直接读写(FC1A在S2入口
 //   2. 自动目标VD584/剩余VD372/累计VD440由引擎直接读写(FC1A在S2入口
//      已初始化,引擎状态0按轮重置VD372=VD584)
 //      已初始化,引擎状态0按轮重置VD372=VD584)
//   3. 错误路径: 引擎内CALL PumpErrExit(FC13A,不变)→停搅拌泵+S_ERROR
 //   3. 错误路径: 引擎内CALL PumpErrExit(FC13A,不变)→停搅拌泵+S_ERROR
// ============================================================
 // ============================================================


END_SUBROUTINE_BLOCK

SUBROUTINE_BLOCK PumpEngine:SBR9
TITLE=// ============================================================
// // 文件: FC23_PumpEngine.stl
// // 功能: 注射泵引擎(v2.5) — 自动/手动共用的完整泵协议状态机
// // 项目: 药液配置与加注控制系统
// // Story: v2.5 注射泵引擎化合并(设计方案见 plc/spec/v2.5_注射泵引擎化合并_设计方案_v1.0.md)
// // PLC: S7-200 SMART CPU ST20
// // 说明: 本文件为语句表(STL)格式，可参考导入STEP 7-Micro/WIN SMART
// //
// // 【v2.5 新建】把原 FC13(自动加药) 与 FC21(手动控制) 中重复实现两遍的
// //   注射泵协议(写指令→等运动→强停→等就绪)抽取为单一引擎:
// //     FC13(自动壳,~35行): 模式=自动 + 搅拌泵断言 + CALL 引擎
// //     FC21(手动壳,~60行): 模式=手动 + HMI镜像 + 启/停命令 + CALL 引擎
// //   根治"两条链路各写一遍必然漂移"的问题(v2.4.1前手动缺强停/缺运动
// //   检测导致"只能吸液"的现场故障即为例证)。
// //
// // 调用关系(互斥,引擎资源共用的安全依据):
// //   自动: OB1 → FC1A(VW418=2) → FC13壳 → CALL PumpEngine
// //   手动: OB1 → FC21壳(VW2=0)  → CALL PumpEngine
// //   两路径永不同扫描周期执行,故 VW226/M11.6/M11.7/M12.0~12.2/T102/T104
// //   全套共用无冲突。
// //
// // 状态表(VW226):
// //   0  初始化/空闲(模式自动: VD372=VD584,VD440不清,跨轮累计;清握手→1。
// //      模式手动: 【v2.5.1】纯空闲不推进, 启动初始化由FC21壳的V307.2
// //      边沿完成(VD372=VD452/VD440=0/清握手)并直接置1——恢复v2.4.1语义,
// //      修复v2.5误把自动语义套用手动导致"无开指令自启动+无限循环"的回归)
// //   1  写抽液(40006=16#9C46;步数=VD372/VD350上限6000;不足一步:
// //      自动→9 / 手动→30)
// //   2  等抽液运动(M12.1开始检测+T102 30s超时;完成/超时→3)
// //   3  强停1(40002=1,无需就绪门控;成功→4)
// //   4  等就绪1(VW4=0;停止请求M13.7→30(仅手动会出现),否则→5)
// //   5  写排液(40007=16#9C47;成功→6)
// //   6  等排液运动(M12.2+T102;完成/超时→7)
// //   7  强停2(40002=1;成功→8)
// //   8  等就绪2+结算(单次扫描: VD440+=VD102×VD350,VD372-=同值;分支:
// //      自动: VD440≥VD584→9,未完成→1;
// //      手动: M13.7→30 / VW388=0单次→30 / VD440≥VD452→30 / 循环未完成→1)
// //   9  完成闩锁(仅自动;清握手+T102;保持闩锁供FC1A消费
// //      "VW226=9 AND T38→VW418=3",转出后由FC1A下轮清VW226)
// //   30 回零(40003=1,仅手动;T102看门狗卡非0态30s→99;门控VW4=0且
// //      VW510=0,或T104冷却到)
// //   40 回零冷却(T104 5s;失败→99;成功→清M13.7/握手→0)
// //   99 错误(仅手动进入;1扫描后自恢复→0)
// //   NET1非法值回收: 合法集{0~9,30,40,99},其余→0+全清
// //
// // 【v2.5.1新增 2026-10-09】泵未就绪自愈块(详见文件体):
// //   引擎在写门控/等就绪状态(1/4/5/8)被VW4≠0(64休眠或100运动中异常残留)
// //   永久阻塞且这些状态无超时。自愈块补发强停(16#9C42,无需就绪门控)把泵
// //   打回96就绪态。64休眠态接受写命令已于2026-10-09现场验证(写强停
// //   VB383=0成功)。上电60s宽限(T105)内不动作, 避免打断泵上电自动复位
// //   (寄存器40026=1, 泵每次上电自检抽排一次, 属正常设备行为)。
// //   完整故障清单见版本库 v2.5.1 提交说明(①~⑤)。
// //
// // 【v2.5.2新增 2026-10-09】状态30两处修复(详见状态30 NETWORK):
// //   ① 滞留写完成清理: M12.0(Done)残留1时 AN M12.0 把状态30写门控永久
// //     锁死, VW226 永久卡30、引擎冻结(现场实锤: VW226=30/M12.0=1 长稳)。
// //     状态30内 M12.0=1 且无写请求/写忙在飞 = 必为残留, 直接清。
// //   ② 回零写门控 "O T104" 修正: 原结构 T104=1 时绕过全部门控每扫描重发
// //     回零; T104 本意仅旁路 VW510 门(写失败冷却重试), 改为草稿位归约。
// //
// // 【v2.5.3新增 2026-10-09】回零重试锁死修复(详见T104 NETWORK):
// //   T104 原仅在状态40驱动, 写失败(VW510>0)后引擎若停在状态30, 门控
// //   (VW510=0 或 T104) 永久锁死(现场实锤: VW510=1 → VW226=30 长稳、
// //   "开"按钮因 VW226≠0 被无视)。扩展为状态30/40双驱动, 冷却5s后重试。
// //
// // 模式位 M17.0 (PumpEngine_ManualMode):
// //   壳每扫描调用引擎前无条件刷新(FC13壳R,FC21壳S),引擎只在被调用
// //   的扫描内读它,无跨扫描持久化问题,冷启动无需专门清零。
// //   OB1"非S0清除"NET按M17.0分流清VW226: 手动中途切自动时清残留子状态
// //   (自动运行期间FC13已把M17.0刷0,清除恒空转,不误伤自动加药)。
// //
// // 符号说明(与FC13/FC21历史版本完全一致,未新增工艺地址):
// // VW226 : 引擎子状态(见状态表;VW390由FC21壳镜像供HMI读取)
// // VD372 : 剩余待加药量(自动=VD584口径,手动=VD452口径;VD396由FC21壳镜像)
// // VD440 : 累计加药量(VD392由FC21壳镜像)
// // VD584 : 自动目标加药量(uL,HMI设定); VD452 : 手动目标加药量(uL,HMI设定)
// // VD350 : 单步分辨率(uL/步); VD102 : 本次循环步数(REAL)
// // VW204/VW206 : 抽/排液步数缓冲(调试查看)
// // VD232/VW230 : FC06写目标地址/数据(FC4任务4消费)
// // M11.6/11.7  : 写请求/写忙(FC4管理); M12.0 : 写完成(FC4置位,引擎清零)
// // M12.1/12.2  : 抽/排液运动已开始(VW4曾=2)
// // M13.7       : 停止请求(仅FC21壳置位,状态4/8消费,状态40成功清除)
// // M17.0       : 模式位(0=自动,1=手动)
// // VW4         : 泵归一化状态码(0=就绪96,1=空闲64,2=运动中100,>=4=错误)
// // V303.4      : 注射泵通讯/动作异常(FC4置位)
// // VW510       : 写任务连续失败计数(FC4管理)
// // T102        : 运动/回零超时(30s); T104 : 回零写冷却(5s)
// // T105        : 【v2.5.1】上电宽限(60s), 泵上电自检期间禁止自愈强停
// // V61.2~V61.7 : 引擎内部条件缓存(引擎总在CALL链最末端执行,不破坏
// //               FC1A在CALL后使用的V61.3)
// // V62.2/V62.3 : 【v2.5.1】自愈块草稿位(全工程检索无冲突; FC21壳的V62.3/
// //               V62.4均在本CALL之前消费完毕, 引擎复用安全)
// // V62.5       : 【v2.5.1】自愈强停在飞闩锁(发强停置位, 消费其写完成后复位)
// // ============================================================
// 
BEGIN
Network 1
//  非法状态自恢复 - 仅回收损坏值(合法集{0~9,30,40,99})
//  各状态前进由T102/V303.4/FC4超时保证,不再需要活动看门狗
//  (v2.4.1 FC21重构时确立的语义,引擎继承)
LDW<   VW226, 0
LDW>   VW226, 9
AW<>   VW226, 30
AW<>   VW226, 40
AW<>   VW226, 99
OLD
=      V61.2
LD     V61.2
MOVW   0, VW226
LD     V61.2
R      M13.7, 1
LD     V61.2
R      M12.0, 3
LD     V61.2
R      M11.6, 2
LD     V61.2
R      T102, 1
LD     V61.2
R      T104, 1
LD     V61.2
R      V62.5, 1              // 【v2.5.1】清自愈强停闩锁(T103写超时会残留)




// 【v2.5.1新增】上电宽限定时器: 泵上电自动复位(设备寄存器40026=1)期间
 // 【v2.5.1新增】上电宽限定时器: 泵上电自动复位(设备寄存器40026=1)期间
//   状态字为100/97等瞬态, 宽限期内禁止自愈块发强停, 避免打断设备自检。
 //   状态字为100/97等瞬态, 宽限期内禁止自愈块发强停, 避免打断设备自检。
//   T105非断电保持, 每次上电从0计60s。
 //   T105非断电保持, 每次上电从0计60s。
LD     Always_On:SM0.0
TON    T105, 600             // 60秒(600×100ms)




// 【v2.5.1新增】泵未就绪自愈块 —— 状态1/4/5/8的写门控/等就绪只认VW4=0,
 // 【v2.5.1新增】泵未就绪自愈块 —— 状态1/4/5/8的写门控/等就绪只认VW4=0,
//   泵若停在64休眠(无误空闲)或100运动异常残留, 这些状态内又无超时,
 //   泵若停在64休眠(无误空闲)或100运动异常残留, 这些状态内又无超时,
//   引擎将永久阻塞(现场实锤: VW4=1卡死手动全流程)。处理: 补发强停
 //   引擎将永久阻塞(现场实锤: VW4=1卡死手动全流程)。处理: 补发强停
//   (16#9C42=1, 无需就绪门控)把泵打回96就绪态, 引擎自然续走。
 //   (16#9C42=1, 无需就绪门控)把泵打回96就绪态, 引擎自然续走。
//   分两段: ①发强停 ②消费这次自愈强停的写完成——必须自家消费,
 //   分两段: ①发强停 ②消费这次自愈强停的写完成——必须自家消费,
//   否则状态1/5的"写成功"分支会误吞该完成信号, 未抽液直跳状态2,
 //   否则状态1/5的"写成功"分支会误吞该完成信号, 未抽液直跳状态2,
//   最终无抽液排液(丢量)。
           //   最终无抽液排液(丢量)。
// 条件: 状态∈{1,4,5,8} AND VW4∈{1,2} AND 无写请求/写忙在飞 AND 宽限外
 // 条件: 状态∈{1,4,5,8} AND VW4∈{1,2} AND 无写请求/写忙在飞 AND 宽限外
LDW=   VW226, 1
LDW=   VW226, 4
OLD
LDW=   VW226, 5
OLD
LDW=   VW226, 8
OLD
AW=    VW4, 1
LDW=   VW4, 2
OLD
AN     M11.6
AN     M11.7
AN     T105
AN     V62.5                 // 上一发自愈强停未完成不重复发
=      V62.2
LD     V62.2
MOVW   1, VW230
MOVD   16#9C42, VD232
S      M11.6, 1
LD     V62.2
S      V62.5, 1              // 闩锁: 自愈强停在飞, 待消费写完成
// 消费段: 自愈强停的写已完成(M11.6已被FC4清)而M12.0仍在→本扫描清掉,
 // 消费段: 自愈强停的写已完成(M11.6已被FC4清)而M12.0仍在→本扫描清掉,
//   不让状态1/3/5/7的成功分支误吞(那些分支针对抽液/排液/强停工序)。
 //   不让状态1/3/5/7的成功分支误吞(那些分支针对抽液/排液/强停工序)。
LD     V62.5
AN     M11.6
A      M12.0
=      V62.3
LD     V62.3
R      M12.0, 1
LD     V62.3
R      V62.5, 1




// 全局错误检测 - 引擎活动期(VW226≠0且≠99)
 // 全局错误检测 - 引擎活动期(VW226≠0且≠99)
// 条件: 活动期 AND (V303.4 OR VW4≥4归一化错误码)
 // 条件: 活动期 AND (V303.4 OR VW4≥4归一化错误码)
// v2.4.1修复门控沿用: VW4=2(运动中)不算错误; V303.4亦要求活动期,
 // v2.4.1修复门控沿用: VW4=2(运动中)不算错误; V303.4亦要求活动期,
//   防止启动瞬间旧报警值误杀新流程(与v2.4.1手动版语义一致;
 //   防止启动瞬间旧报警值误杀新流程(与v2.4.1手动版语义一致;
//   自动路径FC1A在S2入口已R V303.4,此处加闸不改变自动行为)
 //   自动路径FC1A在S2入口已R V303.4,此处加闸不改变自动行为)
LDW<>  VW226, 0
AW<>   VW226, 99
LD     V303.4
LDW<>  VW226, 0
AW<>   VW226, 99
AW>=   VW4, 4
OLD
ALD
=      V61.5
// 自动: 停搅拌泵+转S_ERROR+清子状态(FC13A,现场验证路径,语义不变)
 // 自动: 停搅拌泵+转S_ERROR+清子状态(FC13A,现场验证路径,语义不变)
LD     V61.5
AN     M17.0
CALL   PumpErrExit:SBR27
// 手动: 转99自恢复(报警由V303.4经FC3上报告警画面)
 // 手动: 转99自恢复(报警由V303.4经FC3上报告警画面)
LD     V61.5
A      M17.0
MOVW   99, VW226




// 子状态0 - 初始化(仅自动模式; 手动为纯空闲,见文件头状态表v2.5.1说明)
 // 子状态0 - 初始化(仅自动模式; 手动为纯空闲,见文件头状态表v2.5.1说明)
// 自动: VD372=VD584(VD440不清——FC1A在S2入口已清零,引擎内跨轮累计);
 // 自动: VD372=VD584(VD440不清——FC1A在S2入口已清零,引擎内跨轮累计);
//   清握手→1
                  //   清握手→1
// 【v2.5.1】原"手动: VD372=VD452/VD440=0/清握手→1"分支已删除——它使
 // 【v2.5.1】原"手动: VD372=VD452/VD440=0/清握手→1"分支已删除——它使
//   手动模式状态0无条件自动推进到1, 泵一就绪即自启动打药, 完成后经
 //   手动模式状态0无条件自动推进到1, 泵一就绪即自启动打药, 完成后经
//   30→40→0→1无限循环(v2.5回归, 与v2.4.1空闲语义对比实锤)。手动启动
 //   30→40→0→1无限循环(v2.5回归, 与v2.4.1空闲语义对比实锤)。手动启动
//   初始化改由FC21壳V307.2边沿完成并直接置VW226=1。
 //   初始化改由FC21壳V307.2边沿完成并直接置VW226=1。
LD     Always_On:SM0.0
AW=    VW226, 0
AN     M17.0
=      V61.4
LD     V61.4
MOVR   VD584, VD372
LD     V61.4
R      M12.0, 3
LD     V61.4
R      M11.6, 2
LD     V61.4
R      T102, 1
LD     V61.4
MOVW   1, VW226




// 子状态1 - 计算本次循环步数并下发抽液指令(16#9C46)
 // 子状态1 - 计算本次循环步数并下发抽液指令(16#9C46)
// 条件: 无进行中的写请求/写忙/写完成
      // 条件: 无进行中的写请求/写忙/写完成
// 【2026-10-08修复 v2.3.9】ROUND后DTR(原MOVR位拷贝按REAL解读为
 // 【2026-10-08修复 v2.3.9】ROUND后DTR(原MOVR位拷贝按REAL解读为
//   denormal≈0,步数蒸发→恒判"不足一步")
 //   denormal≈0,步数蒸发→恒判"不足一步")
LD     Always_On:SM0.0
AW=    VW226, 1
AN     M11.6
AN     M11.7
AN     M12.0
MOVR   VD372, VD102
/R     VD350, VD102
ROUND  VD102, AC0
DTR    AC0, VD102
// 限制最大6000步(25ml注射器容量),先ROUND/DTR后比较覆盖(v2.4.0)
 // 限制最大6000步(25ml注射器容量),先ROUND/DTR后比较覆盖(v2.4.0)
LD     Always_On:SM0.0
AR>=   VD102, 6000.0
MOVR   6000.0, VD102
// 检查步数有效性(不足一步直接完成)
        // 检查步数有效性(不足一步直接完成)
LD     Always_On:SM0.0
AR<=   VD102, 0.0
JMP    22
ROUND  VD102, AC0
// 同步写入抽/排液步数缓冲(供HMI/调试查看)
  // 同步写入抽/排液步数缓冲(供HMI/调试查看)
MOVW   AC0, VW204
MOVW   AC0, VW206
// 重新建立执行条件后下发抽液指令
          // 重新建立执行条件后下发抽液指令
// ★泵就绪(VW4=0)才允许写, 避免运动中下发导致异常码4
 // ★泵就绪(VW4=0)才允许写, 避免运动中下发导致异常码4
LD     Always_On:SM0.0
AW=    VW226, 1
AN     M11.6
AN     M11.7
AN     M12.0
AW=    VW4, 0
MOVW   AC0, VW230
MOVD   16#9C46, VD232
S      M11.6, 1
JMP    23
LBL    22
// 剩余量不足一步,无需再加药
            // 剩余量不足一步,无需再加药
// 自动→9(完成闩锁); 手动→30(回零)
    // 自动→9(完成闩锁); 手动→30(回零)
LD     M17.0
MOVW   30, VW226
LD     M17.0
NOT
MOVW   9, VW226
LBL    23




// 子状态1/5 - 写完成处理(抽液/排液共享,错误路径按模式分流)
 // 子状态1/5 - 写完成处理(抽液/排液共享,错误路径按模式分流)
// 错误: 子状态1或5 + V303.4(写失败)
 // 错误: 子状态1或5 + V303.4(写失败)
LD     M12.0
LD     Always_On:SM0.0
AW=    VW226, 1
LD     Always_On:SM0.0
AW=    VW226, 5
OLD
A      V303.4
=      V61.2
LD     V61.2
AN     M17.0
CALL   PumpErrExit:SBR27
LD     V61.2
A      M17.0
MOVW   99, VW226
// 成功: 子状态1→2(抽液写成功 → 等抽液运动完成)
 // 成功: 子状态1→2(抽液写成功 → 等抽液运动完成)
LD     M12.0
AW=    VW226, 1
AN     V303.4
R      M12.0, 1
R      M11.6, 1
MOVW   2, VW226
// 成功: 子状态5→6(排液写成功 → 等排液运动完成)
 // 成功: 子状态5→6(排液写成功 → 等排液运动完成)
LD     M12.0
AW=    VW226, 5
AN     V303.4
R      M12.0, 1
R      M11.6, 1
MOVW   6, VW226




// 子状态2/6 - 等待运动完成(抽液M12.1/排液M12.2)
 // 子状态2/6 - 等待运动完成(抽液M12.1/排液M12.2)
// T102: 30秒超时(防止泵卡在运动态),子状态2/6复用
 // T102: 30秒超时(防止泵卡在运动态),子状态2/6复用
// 完成: (M12.x=1 AND VW4≠2) OR T102超时 → 子状态3/7(写强停)
 // 完成: (M12.x=1 AND VW4≠2) OR T102超时 → 子状态3/7(写强停)
// 运动检测: VW4=2(100运动中)→M12.x置位,VW4≠2且已开始→运动完成
 // 运动检测: VW4=2(100运动中)→M12.x置位,VW4≠2且已开始→运动完成


// T102运行(子状态2/6/30) —— 【v2.5.1修复】原"2/6"与"30"两处NETWORK
 // T102运行(子状态2/6/30) —— 【v2.5.1修复】原"2/6"与"30"两处NETWORK
//   分别驱动同一T102, 同扫描内后执行NETWORK把先执行者复位, T102永不
 //   分别驱动同一T102, 同扫描内后执行NETWORK把先执行者复位, T102永不
//   计满→运动超时与回零看门狗双双失效(现场实锤: 状态30冻结1小时无超时)。
 //   计满→运动超时与回零看门狗双双失效(现场实锤: 状态30冻结1小时无超时)。
//   合并为单一NETWORK驱动, 三态共用30s(语义不变: 2/6超时→强停恢复,
 //   合并为单一NETWORK驱动, 三态共用30s(语义不变: 2/6超时→强停恢复,
//   30超时→99)。
              //   30超时→99)。
LD     Always_On:SM0.0
AW=    VW226, 2
LD     Always_On:SM0.0
AW=    VW226, 6
OLD
LD     Always_On:SM0.0
AW=    VW226, 30
OLD
TON    T102, 300             // 30秒(300×100ms)


// 检测运动开始: 子状态2
             // 检测运动开始: 子状态2
LD     Always_On:SM0.0
AW=    VW226, 2
AW=    VW4, 2
S      M12.1, 1
// 检测运动开始: 子状态6
             // 检测运动开始: 子状态6
LD     Always_On:SM0.0
AW=    VW226, 6
AW=    VW4, 2
S      M12.2, 1


// 运动完成: 子状态2→3(写强停恢复)
      // 运动完成: 子状态2→3(写强停恢复)
LD     M12.1
AW=    VW226, 2
AW<>   VW4, 2
R      T102, 1
R      M12.1, 1
MOVW   3, VW226


// 运动完成: 子状态6→7(写强停恢复)
      // 运动完成: 子状态6→7(写强停恢复)
LD     M12.2
AW=    VW226, 6
AW<>   VW4, 2
R      T102, 1
R      M12.2, 1
MOVW   7, VW226


// 超时: 子状态2→3(强停恢复,防止卡死,不报错——同FC13策略)
 // 超时: 子状态2→3(强停恢复,防止卡死,不报错——同FC13策略)
LD     T102
AW=    VW226, 2
R      T102, 1
R      M12.1, 1
MOVW   3, VW226


// 超时: 子状态6→7
               // 超时: 子状态6→7
LD     T102
AW=    VW226, 6
R      T102, 1
R      M12.2, 1
MOVW   7, VW226




// 子状态3/7 - 下发强停指令(16#9C42=1)恢复96就绪
 // 子状态3/7 - 下发强停指令(16#9C42=1)恢复96就绪
// ★强停无需就绪门控: 用于紧急停止/恢复, 不检查VW4=0
 // ★强停无需就绪门控: 用于紧急停止/恢复, 不检查VW4=0
LD     Always_On:SM0.0
AW=    VW226, 3
LD     Always_On:SM0.0
AW=    VW226, 7
OLD
AN     M11.6
AN     M11.7
AN     M12.0
LPS
MOVW   1, VW230              // 强停数据=1
MOVD   16#9C42, VD232        // ★十六进制地址(40002=16#9C42)
S      M11.6, 1              // 置写请求
LPP




// 子状态3/7 - 强停写完成处理(共享错误路径,按模式分流)
 // 子状态3/7 - 强停写完成处理(共享错误路径,按模式分流)
LD     M12.0
LD     Always_On:SM0.0
AW=    VW226, 3
LD     Always_On:SM0.0
AW=    VW226, 7
OLD
A      V303.4
=      V61.2
LD     V61.2
AN     M17.0
CALL   PumpErrExit:SBR27
LD     V61.2
A      M17.0
MOVW   99, VW226
// 成功: 子状态3→4(等强停完成+恢复就绪)
   // 成功: 子状态3→4(等强停完成+恢复就绪)
LD     M12.0
AW=    VW226, 3
AN     V303.4
R      M12.0, 1
R      M11.6, 1
MOVW   4, VW226
// 成功: 子状态7→8(等强停完成+结算)
     // 成功: 子状态7→8(等强停完成+结算)
LD     M12.0
AW=    VW226, 7
AN     V303.4
R      M12.0, 1
R      M11.6, 1
MOVW   8, VW226




// 子状态4 - 等待泵恢复就绪(VW4=0=96就绪态),消费停止请求
 // 子状态4 - 等待泵恢复就绪(VW4=0=96就绪态),消费停止请求
// 强停后泵从100→96, 需等待VW4回到0才能接受下一条命令
 // 强停后泵从100→96, 需等待VW4回到0才能接受下一条命令
// 停止请求M13.7仅手动壳可置位(自动路径恒走"→5"分支,无需模式门控)
 // 停止请求M13.7仅手动壳可置位(自动路径恒走"→5"分支,无需模式门控)
LD     Always_On:SM0.0
AW=    VW226, 4
AW=    VW4, 0
AN     M13.7
MOVW   5, VW226              // 正常→写排液
LD     Always_On:SM0.0
AW=    VW226, 4
AW=    VW4, 0
A      M13.7
MOVW   30, VW226             // 停止请求→回零




// 子状态5 - 下发排液指令(16#9C47)
   // 子状态5 - 下发排液指令(16#9C47)
// ★泵就绪(VW4=0)才允许写, 避免运动中下发导致异常码4
 // ★泵就绪(VW4=0)才允许写, 避免运动中下发导致异常码4
LD     Always_On:SM0.0
AW=    VW226, 5
AN     M11.6
AN     M11.7
AN     M12.0
AW=    VW4, 0
LPS
ROUND  VD102, AC0
MOVW   AC0, VW230
MOVW   AC0, VW206
MOVD   16#9C47, VD232        // ★十六进制地址(40007=16#9C47)
S      M11.6, 1
LPP




// 子状态8 - 等待泵恢复就绪 + 计算本轮体积 + 模式分支(全部同扫描完成)
 // 子状态8 - 等待泵恢复就绪 + 计算本轮体积 + 模式分支(全部同扫描完成)
// 等待VW4=0(就绪), 然后计算本轮排出药量, 按模式分流:
 // 等待VW4=0(就绪), 然后计算本轮排出药量, 按模式分流:
//   自动(M17.0=0): VD440≥VD584→9(完成闩锁); 未完成→1(下一轮)
 //   自动(M17.0=0): VD440≥VD584→9(完成闩锁); 未完成→1(下一轮)
//   手动(M17.0=1): M13.7→30(停止); VW388=0单次→30;
 //   手动(M17.0=1): M13.7→30(停止); VW388=0单次→30;
//                  VD440≥VD452→30(循环完成); 否则→1(循环下一轮)
 //                  VD440≥VD452→30(循环完成); 否则→1(循环下一轮)
// 同扫描分支保证结算只执行一次
           // 同扫描分支保证结算只执行一次
LD     Always_On:SM0.0
AW=    VW226, 8
AW=    VW4, 0
=      V61.6
// 计算本次循环实际排出药量 = VD102 × VD350, 累加/扣减
 // 计算本次循环实际排出药量 = VD102 × VD350, 累加/扣减
LD     V61.6
MOVR   VD102, AC0            // AC0 = 本次循环步数(REAL)
LD     V61.6
*R     VD350, AC0            // AC0 = 本次循环体积(μL)
LD     V61.6
+R     AC0, VD440            // 累计加药量 += 本次循环体积
LD     V61.6
-R     AC0, VD372            // 剩余量 -= 本次循环体积
LD     V61.6
R      M12.0, 3
LD     V61.6
R      M11.6, 2
// 自动: 完成→9闩锁
               // 自动: 完成→9闩锁
LD     V61.6
AN     M17.0
AR>=   VD440, VD584
MOVW   9, VW226
// 自动: 未完成→下一轮
              // 自动: 未完成→下一轮
LD     V61.6
AN     M17.0
AR<    VD440, VD584
MOVW   1, VW226
// 手动: 停止请求→回零(优先级最高,分支置于单次/循环之前判定)
 // 手动: 停止请求→回零(优先级最高,分支置于单次/循环之前判定)
LD     V61.6
A      M17.0
A      M13.7
MOVW   30, VW226
// 手动: 单次模式→回零
              // 手动: 单次模式→回零
LD     V61.6
A      M17.0
AW=    VW388, 0
MOVW   30, VW226
// 手动: 循环模式且累计≥目标→回零
        // 手动: 循环模式且累计≥目标→回零
LD     V61.6
A      M17.0
AW=    VW388, 1
AR>=   VD440, VD452
MOVW   30, VW226
// 手动: 循环模式且未完成(且无停止请求)→下一轮
 // 手动: 循环模式且未完成(且无停止请求)→下一轮
LD     V61.6
A      M17.0
AN     M13.7
AW=    VW388, 1
AR<    VD440, VD452
MOVW   1, VW226




// 子状态9 - 完成闩锁(仅自动路径进入)
     // 子状态9 - 完成闩锁(仅自动路径进入)
// 清握手+停运动超时, **保持VW226=9作"加药完成"闩锁**
 // 清握手+停运动超时, **保持VW226=9作"加药完成"闩锁**
// (v2.3.4修订语义: FC1A看到"9+T38到"→VW418=3转出S2; 下轮S2由FC1A
 // (v2.3.4修订语义: FC1A看到"9+T38到"→VW418=3转出S2; 下轮S2由FC1A
//   首次进入清VW226=0,语义闭环。手动完成走30回零,不进9)
 //   首次进入清VW226=0,语义闭环。手动完成走30回零,不进9)
LD     Always_On:SM0.0
AW=    VW226, 9
R      M12.0, 3
R      M11.6, 2
R      T102, 1




// 子状态30 - 回零(40003=1,仅手动路径进入;活塞归零)
 // 子状态30 - 回零(40003=1,仅手动路径进入;活塞归零)
// T102兼作回零看门狗——泵若卡非0态(VW4≠0),30秒后转99,不再无限等待
 // T102兼作回零看门狗——泵若卡非0态(VW4≠0),30秒后转99,不再无限等待
// 【v2.5.1】T102驱动已合并至上方"子状态2/6/30"单一NETWORK, 此处仅取超时
 // 【v2.5.1】T102驱动已合并至上方"子状态2/6/30"单一NETWORK, 此处仅取超时
LD     T102
AW=    VW226, 30
MOVW   99, VW226
// 【v2.5.2新增】状态30滞留写完成清理——状态30内 M12.0=1 且无写请求/写忙
 // 【v2.5.2新增】状态30滞留写完成清理——状态30内 M12.0=1 且无写请求/写忙
//   在飞 = 滞留的 Done 位。正常流程状态30发命令同扫描即转40, 写完成由
 //   在飞 = 滞留的 Done 位。正常流程状态30发命令同扫描即转40, 写完成由
//   状态40消费, 所以状态30见到 M12.0=1 必然是残留(手动置M11.6调试/
 //   状态40消费, 所以状态30见到 M12.0=1 必然是残留(手动置M11.6调试/
//   停止命令打断在飞写/断电恢复等)。不清则 AN M12.0 把下方写门控永久
 //   停止命令打断在飞写/断电恢复等)。不清则 AN M12.0 把下方写门控永久
//   锁死, VW226 永久卡30、引擎冻结(现场实锤: VW226=30/M12.0=1 长时间
 //   锁死, VW226 永久卡30、引擎冻结(现场实锤: VW226=30/M12.0=1 长时间
//   稳定不动)。清理后写门控按 VW4=0 自然打开, 引擎正常 30→40→0 收尾。
 //   稳定不动)。清理后写门控按 VW4=0 自然打开, 引擎正常 30→40→0 收尾。
LD     Always_On:SM0.0
AW=    VW226, 30
AN     M11.6
AN     M11.7
A      M12.0
R      M12.0, 1
// 写回零指令(VW510连续写失败时等T104冷却重试)
 // 写回零指令(VW510连续写失败时等T104冷却重试)
// 【v2.5.2修复】原 "AW= VW510,0 / O T104" 把 T104 挂在整条AND链之外,
 // 【v2.5.2修复】原 "AW= VW510,0 / O T104" 把 T104 挂在整条AND链之外,
//   T104=1 时会无视 M11.6/M11.7/M12.0/VW4=0 每扫描重发回零。T104 的本意
 //   T104=1 时会无视 M11.6/M11.7/M12.0/VW4=0 每扫描重发回零。T104 的本意
//   仅是"VW510>0 写连续失败时, 冷却5秒后允许重试"——只应旁路 VW510 门控,
 //   仅是"VW510>0 写连续失败时, 冷却5秒后允许重试"——只应旁路 VW510 门控,
//   改为先用草稿位 V61.4 归约 (VW510=0 OR T104) 再并入主链。
 //   改为先用草稿位 V61.4 归约 (VW510=0 OR T104) 再并入主链。
LDW=   VW510, 0
O      T104
=      V61.4
LD     Always_On:SM0.0
AW=    VW226, 30
AN     M11.6
AN     M11.7
AN     M12.0
AW=    VW4, 0
A      V61.4
MOVW   1, VW230
MOVD   16#9C43, VD232        // ★十六进制地址(40003=16#9C43)
S      M11.6, 1
MOVW   40, VW226




// T104冷却定时器(回零写连续失败时,5秒后允许重试)
 // T104冷却定时器(回零写连续失败时,5秒后允许重试)
// 【v2.5.3修复】原仅在状态40驱动: 写请求若在状态30发出后失败且引擎回到
 // 【v2.5.3修复】原仅在状态40驱动: 写请求若在状态30发出后失败且引擎回到
//   状态30(VW510>0), 状态30内T104永不驱动→门控(VW510=0或T104)永久锁死,
 //   状态30(VW510>0), 状态30内T104永不驱动→门控(VW510=0或T104)永久锁死,
//   VW226永久卡30(现场实锤: VW510=1时VW226=30长稳、回零写被挡)。
 //   VW226永久卡30(现场实锤: VW510=1时VW226=30长稳、回零写被挡)。
//   扩展为状态30/40均可驱动: 状态30内VW510>0时冷却5s后由T104旁路VW510门
 //   扩展为状态30/40均可驱动: 状态30内VW510>0时冷却5s后由T104旁路VW510门
//   重试; 写一发出门控段即离开状态30, T104自然复位, 不会连发。
 //   重试; 写一发出门控段即离开状态30, T104自然复位, 不会连发。
LD     M12.0
AW=    VW226, 40
AW>    VW510, 0
LD     Always_On:SM0.0
AW=    VW226, 30
AW>    VW510, 0
OLD
TON    T104, 50              // 5秒(50×100ms)




// 子状态40 - 回零写完成处理
          // 子状态40 - 回零写完成处理
// 失败→99(错误自恢复); 成功→清停止请求及握手→回空闲0
 // 失败→99(错误自恢复); 成功→清停止请求及握手→回空闲0
LD     M12.0
AW=    VW226, 40
A      V303.4
MOVW   99, VW226
LD     M12.0
AW=    VW226, 40
AN     V303.4
R      M12.0, 1
R      M13.7, 1
R      M11.6, 2
R      T104, 1
R      T102, 1
MOVW   0, VW226




// 子状态99 - 错误自恢复(1扫描后回0,仅手动路径进入)
 // 子状态99 - 错误自恢复(1扫描后回0,仅手动路径进入)
// 自动错误直接走PumpErrExit转S_ERROR,不进99
 // 自动错误直接走PumpErrExit转S_ERROR,不进99
// 报警可见性由V303.4经FC3报警画面保证
   // 报警可见性由V303.4经FC3报警画面保证
LDW=   VW226, 99
=      V61.7
LD     V61.7
R      M13.7, 1
LD     V61.7
R      M12.0, 3
LD     V61.7
R      M11.6, 2
LD     V61.7
R      T102, 1
LD     V61.7
R      T104, 1
LD     V61.7
R      V62.5, 1              // 【v2.5.1】清自愈强停闩锁
LD     V61.7
MOVW   0, VW226




// ============================================================
 // ============================================================
// 文件结束
                     // 文件结束
// 说明:
                      // 说明:
//   1. 全流程泵协议: 抽液→等运动→强停→等就绪→排液→等运动→强停→等就绪
 //   1. 全流程泵协议: 抽液→等运动→强停→等就绪→排液→等运动→强停→等就绪
//      →结算/循环,每段运动后必发强停(40002=1)恢复96就绪态
 //      →结算/循环,每段运动后必发强停(40002=1)恢复96就绪态
//   2. 运动检测: VW4=2→M12.x置位; VW4≠2且M12.x=1→完成; T102(30s)超时
 //   2. 运动检测: VW4=2→M12.x置位; VW4≠2且M12.x=1→完成; T102(30s)超时
//      走强停恢复不报错(泵可能未完成动作,与FC13历史口径一致)
 //      走强停恢复不报错(泵可能未完成动作,与FC13历史口径一致)
//   3. 引擎内停止检查(M13.7)无模式门控: M13.7只能由FC21壳置位,
 //   3. 引擎内停止检查(M13.7)无模式门控: M13.7只能由FC21壳置位,
//      OB1离S0即清,自动路径物理上不可能置位
 //      OB1离S0即清,自动路径物理上不可能置位
//   4. V位缓存V61.2~V61.7仅引擎使用; FC1A在CALL FC13后会用V61.3,
 //   4. V位缓存V61.2~V61.7仅引擎使用; FC1A在CALL FC13后会用V61.3,
//      引擎避开V61.3(调用链: FC1A→FC13→引擎,引擎总在末端)
 //      引擎避开V61.3(调用链: FC1A→FC13→引擎,引擎总在末端)
//   5. 所有Modbus地址使用十六进制格式(16#9C46/16#9C47/16#9C42/16#9C43)
 //   5. 所有Modbus地址使用十六进制格式(16#9C46/16#9C47/16#9C42/16#9C43)
//      避免十进制大数被解析为INT导致MBUS_MSG Error=6
 //      避免十进制大数被解析为INT导致MBUS_MSG Error=6
//   6. JMP/LBL(22/23)在本NETWORK内,无跨NETWORK跳转问题(问题#21教训)
 //   6. JMP/LBL(22/23)在本NETWORK内,无跨NETWORK跳转问题(问题#21教训)
//   7.【v2.5.1】T102仅"子状态2/6/30"一处NETWORK驱动, 禁止再添加第二处
 //   7.【v2.5.1】T102仅"子状态2/6/30"一处NETWORK驱动, 禁止再添加第二处
//      驱动点(重复驱动=同扫描互复位=看门狗静默失效, 现场冻结1小时实锤)
 //      驱动点(重复驱动=同扫描互复位=看门狗静默失效, 现场冻结1小时实锤)
//   8.【v2.5.1】自愈块与全局错误块顺序: 自愈消费段在前, 保证自愈强停的
 //   8.【v2.5.1】自愈块与全局错误块顺序: 自愈消费段在前, 保证自愈强停的
//      写完成被自家清掉, 不被状态1/3/5/7成功分支误吞
 //      写完成被自家清掉, 不被状态1/3/5/7成功分支误吞
//   9.【v2.5.2】状态30滞留 M12.0 清理网络置于写门控之前, 且只在
 //   9.【v2.5.2】状态30滞留 M12.0 清理网络置于写门控之前, 且只在
//      M11.6=M11.7=0(无在飞写)时清, 绝不误吞真正在飞的写完成
 //      M11.6=M11.7=0(无在飞写)时清, 绝不误吞真正在飞的写完成
// ============================================================
 // ============================================================


END_SUBROUTINE_BLOCK

SUBROUTINE_BLOCK State_S4_Transfer:SBR10
TITLE=// ============================================================
// // 文件: FC15_State_S4_Transfer.stl
// // 功能: S4上→下转移 (VW2=5)
// // Story: v2.2 流程重构 (替代 AQEX-6 状态机骨架 + AQEX-7 阀门诊断)
// // 说明: v2.2 S4 是唯一的上下缸交汇点
// //       启动条件: VW2=5 AND V1.7=0 (下缸已排空) AND VW418=3 (上缸已配完)
// //       完成后: 切 VW418=4 (已转移) + 写 S6 滚动默认值 + 转 S5
// // ============================================================
BEGIN
Network 1
//  S4 启动条件(v2.2 关键改动:必须 VW418=3 才能启动)
//  触发条件: VW2=5 (下缸 S4 入口) + V1.7=0 (下缸已排空) + VW418=3 (上缸配完等待) + VW6=0 (无报警)
//  启动动作: 开阀B + 启动 T49 计时 + 置 VW418=4 (上缸标记"已转移")
//  【v10.4硬件变更】下缸NC球阀Q0.6已去除(保留未使用),不再随S4启动
//  [已修复 v2.2] 用 V61.5 缓存 S4 启动条件,避免 LPS/LPP+NOT 配合下的 S/R 链栈空
//  【v2.3修复】首轮补入口: 下缸S5空等(VW2=6)且已排空(V1.7=0)且上缸已配完(VW418=3)
//    原仅响应VW2=5,首轮FC10直接置VW2=6,首罐液体永远无法转移
LD     Always_On:SM0.0       // S4 状态入口
AW=    VW2, 5                // 下缸已排空
AN     V1.7                  // 上缸已配完
AW=    VW418, 3              // 无报警
=      V61.5
AW=    VW6, 0                // 【v2.3】首轮入口(VW2=6空等,条件与上面等价)
AW=    VW2, 6
AN     V1.7
AW=    VW418, 3
AW=    VW6, 0
=      V61.5                 // 两个入口取或
=      V61.5
LDN    V61.5
LD     Always_On:SM0.0       // 任一条件不满足 → 不启动
// 条件满足 → 启动 S4 转液           // 条件满足 → 启动 S4 转液
LD     V61.5
AW=    VW2, 6                // 开阀B
LD     V61.5
R      T49, 1
LD     SM0.0
AN     V1.7                  // 【v2.3修复】S4 实测计时,PT=VW288独立地址
                                   // (原VW290被FC4 Modbus任务状态机占用,每周期改写,计时不确定) // (原VW290被FC4 Modbus任务状态机占用,每周期改写,计时不确定)
// 置 VW418=4 (上缸已转移)         // 置 VW418=4 (上缸已转移)
LD     V61.5
MOVW   4, VW418
JMP    2
LBL    1
LBL    2
// 注: 条件不满足时 S/R/计时/赋值指令全部不执行, FC31 诊断空转, 等待下一周期 // 注: 条件不满足时 S/R/计时/赋值指令全部不执行, FC31 诊断空转, 等待下一周期
// 【v2.2 兼容保留】S4 等待超时逻辑(下缸未排空时使用) // 【v2.2 兼容保留】S4 等待超时逻辑(下缸未排空时使用)
// [已修复 v2.2] 用 V61.6 缓存 S4 等待条件,避免 LPS/LPP+NOT 配合下的栈空 // [已修复 v2.2] 用 V61.6 缓存 S4 等待条件,避免 LPS/LPP+NOT 配合下的栈空
// v2.2 仍保留 V303.2 报警机制(仅提示不强制 S_ERROR) // v2.2 仍保留 V303.2 报警机制(仅提示不强制 S_ERROR)
// 与 v2.1 区别: 增加"上缸配完"判断(原版只看 V1.7) // 与 v2.1 区别: 增加"上缸配完"判断(原版只看 V1.7)
LD     SM0.0
AW=    VW2, 5
// 启动条件:V1.7=1(下缸未空) AND VW418=3(上缸配完) // 启动条件:V1.7=1(下缸未空) AND VW418=3(上缸配完)
A      V1.7
AW=    VW418, 3
=      V61.6
LDN    V61.6
JMP    3
// 下缸未空,启动 T61 等待计时          // 下缸未空,启动 T61 等待计时
LD     V61.6
AW=    VW418, 3              // VD_S4WaitTimeout
*R     10.0, VD324
ROUND  VD324, AC0
AW=    VW6, 0                // T61 PT
LD     V61.6
R      T61, 1
LD     SM0.0
O      V61.5                 // S4 等待超时计时
// 每秒累加 VD_S4Wait_Time (T62 1s 脉冲) // 每秒累加 VD_S4Wait_Time (T62 1s 脉冲)
LD     V61.6
R      T62, 1
LD     SM0.0
TON    T62, 10
LD     T62
EU
=      V61.5                 // VD_S4Wait_Time + 1s
R      T62, 1
// 超时报警                      // 超时报警
LD     T61
LDN    V61.5                 // M_Alarm_S4TransferWaitTimeout
JMP    4
LBL    3
LBL    4
// 调用阀B诊断                    // 调用阀B诊断
LD     SM0.0
CALL ValveB_Diag
// 检查阀B诊断结果 + S4 完成动作        // 检查阀B诊断结果 + S4 完成动作
// [已修复 v2.2] 用 V61.7 缓存诊断完成条件,避免 LPS/LPP+NOT 配合下的 S/R 链栈空 // [已修复 v2.2] 用 V61.7 缓存诊断完成条件,避免 LPS/LPP+NOT 配合下的 S/R 链栈空
// v2.2 关键改动:完成时切 M16.0 = NOT M16.0(双倒计时器切换),写 VD116 (S6_actual 滚动) // v2.2 关键改动:完成时切 M16.0 = NOT M16.0(双倒计时器切换),写 VD116 (S6_actual 滚动)
//   注: 首轮时 VD116 存 S4 实测时长,后续轮次存 S6 实测时长(用于 FC40 S6 触发阈值) //   注: 首轮时 VD116 存 S4 实测时长,后续轮次存 S6 实测时长(用于 FC40 S6 触发阈值)
LD     SM0.0
JMP    1                     // 阀B诊断正常完成(VB268=1)
=      V61.7
LDN    V61.7
LD     V61.5                 // 未完成 → 跳到 NETWORK 4 末尾
// 诊断完成 → 执行 S4 完成动作         // 诊断完成 → 执行 S4 完成动作
// 【v2.3修复】先读T49当前值再复位(R在前读到的恒为0) // 【v2.3修复】先读T49当前值再复位(R在前读到的恒为0)
LD     V61.7
S      CPU_输出3:Q0.3, 1       // T49 当前值(100ms 时基)
LD     V61.5                 // → DINT
DTR    VD444, VD444
R      T49, 1                // 【v2.3.6】100ms时基→秒                // → REAL(原值秒)
LD     Always_On:SM0.0       // VD116 = S4 实测秒(首轮作 S6 默认)
LD     V61.7
R      T49, 1
// 置下缸状态=满                   // 置下缸状态=满
LD     V61.7
S      V1.7, 1
// 记录下缸变满时间戳                 // 记录下缸变满时间戳
LD     V61.7
TODR   VB900
MOVB   VB900, VB10
MOVB   VB901, VB11
MOVB   VB902, VB12
MOVB   VB903, VB13
MOVB   VB904, VB14
MOVB   VB905, VB15
MOVB   VB906, VB16
MOVB   VB908, VB17
// 下缸实验时长清零                  // 下缸实验时长清零
LD     V61.7
TON    T49, VW288            // VD_S5_Elapsed 清零
LD     V61.7
LD     V61.5                 // 清预规划标志
// S4 等待计时清零                 // S4 等待计时清零
LD     V61.7
MOVW   4, VW418              // 清 T61+T62 (连续2个定时器)
LD     V61.7
JMP    2                     // VD_S4Wait_Time 清零(恢复原始中间变量用途)
LD     V61.7
LBL    1                     // 清 S4 等待超时报警
// 【v2.3删除】原"切双倒计时器标记 M16.0 = NOT M16.0"已删: // 【v2.3删除】原"切双倒计时器标记 M16.0 = NOT M16.0"已删:
//   M16.0 全程序仅在 FC17 S6 完成时切换一次(原S4/S6各切一次导致每周期翻转两次) //   M16.0 全程序仅在 FC17 S6 完成时切换一次(原S4/S6各切一次导致每周期翻转两次)
// 【v2.3删除】原"触发下一轮 S1 脉冲 S M16.1"已删: // 【v2.3删除】原"触发下一轮 S1 脉冲 S M16.1"已删:
//   下一轮 S1 由 FC40 按 Elapsed>=T_cycle-Prep_Needed 触发(VW418=4 门控); //   下一轮 S1 由 FC40 按 Elapsed>=T_cycle-Prep_Needed 触发(VW418=4 门控);
//   此处置位会使上缸刚置"已转移"就立即启动下一轮,破坏24h周期约束 //   此处置位会使上缸刚置"已转移"就立即启动下一轮,破坏24h周期约束
// 状态转移 S4→S5                // 状态转移 S4→S5
LD     V61.7
MOVW   6, VW2
LBL    10
// 注: 漫溢保护、四态诊断、开关到位、超时保护全部由 FC31 统一处理 // 注: 漫溢保护、四态诊断、开关到位、超时保护全部由 FC31 统一处理
// 注: 【v10.4硬件变更】下缸NC球阀已去除,FC31漫溢保护仅关阀B,不再操作Q0.6 // 注: 【v10.4硬件变更】下缸NC球阀已去除,FC31漫溢保护仅关阀B,不再操作Q0.6
// 注: DT 时间戳格式需与 S7-200 SMART 的 DT 数据类型对齐 // 注: DT 时间戳格式需与 S7-200 SMART 的 DT 数据类型对齐
// 注: 断电恢复由 FC0 统一处理,VW2=5 (S4 阀B动作中断) 时 FC0 转 S_ERROR // 注: 断电恢复由 FC0 统一处理,VW2=5 (S4 阀B动作中断) 时 FC0 转 S_ERROR
// ============================================================ // ============================================================
// 文件结束                      // 文件结束
// ============================================================

 // ============================================================
LBL    2
LD     Always_On:SM0.0
AW=    VW2, 5
A      V1.7
AW=    VW418, 3
=      V61.6
LDN    V61.6
JMP    3
LD     V61.6
MOVR   VD448, VD324
*R     10.0, VD324
ROUND  VD324, AC0
MOVW   AC0, VW286
LD     V61.6
R      T61, 1
LD     Always_On:SM0.0
TON    T61, VW286
LD     V61.6
R      T62, 1
LD     Always_On:SM0.0
TON    T62, 10
LD     T62
EU
+R     1.0, VD444
R      T62, 1
LD     T61
S      V303.2, 1
JMP    4
LBL    3
LBL    4
LD     Always_On:SM0.0
CALL   ValveB_Diag:SBR17
LD     Always_On:SM0.0
AB=    VB268, 1
=      V61.7
LDN    V61.7
JMP    10
LD     V61.7
MOVW   T49, AC0
ITD    AC0, VD444
DTR    VD444, VD444
/R     10.0, VD444
MOVR   VD444, VD116
LD     V61.7
R      T49, 1
LD     V61.7
S      V1.7, 1
LD     V61.7
TODR   VB900
MOVB   VB900, VB10
MOVB   VB901, VB11
MOVB   VB902, VB12
MOVB   VB903, VB13
MOVB   VB904, VB14
MOVB   VB905, VB15
MOVB   VB906, VB16
MOVB   VB908, VB17
LD     V61.7
MOVR   0.0, VD178
LD     V61.7
R      M10.7, 1
LD     V61.7
R      T61, 2
LD     V61.7
MOVR   0.0, VD444
LD     V61.7
R      V303.2, 1
LD     V61.7
MOVW   6, VW2
LBL    10
END_SUBROUTINE_BLOCK

SUBROUTINE_BLOCK State_S5_Run:SBR11
TITLE=// ============================================================
// // 文件: FC16_State_S5_Run.stl
// // 功能: S5 实验运行中 (VW2=6)
// // Story: v2.2 流程重构 (替代 AQEX-6 状态机骨架 + AQEX-8 节奏纠偏)
// // 说明: v2.2 S5 仅负责:
// //       1. 下缸满计时 VD_S5_Elapsed 累加
// //       2. 实验时长累加 VD_ExperimentDuration_Accum
// //       3. 换水周期到达转 S6 (VD_S5_Elapsed >= 阈值, 阈值 = 86400/VD414 - VD426 - VD430)
// //       4. 实验时长达标转 S7
// //   v2.2 删除:
// //       - 原三层纠偏预规划 (VD_CycleSetpoint×60 触发)
// //       - 启动 VW2=1 (上缸配液) 触发逻辑 (改由 FC40 触发下一轮 S1)
// //       - VD354 / VW182 / VW184 / VD112 / VD150 / VD154 引用
// //       - M10.7 预规划标志 (改由 FC40 M16.1 替代)
// // ============================================================
// 
BEGIN
Network 1
//  [已修复 v2.2] 删除 VD178 累加逻辑,统一由 FC40 双倒计时器管理周期
//  注: VD178 保留清零/初始化,仅作兼容显示,不再参与控制
//  实验时长累加(仅下缸=满期间,每分钟+1)
//  VD_ExperimentDuration_Accum(VD366)每分钟+1
LD     Clock_60s:SM0.4       // 系统分时钟(1min周期)
A      V1.7                  // 且下缸=满
EU                           // 【v2.3.6修复2026-09-30】每满1分钟一脉冲; 原T47每扫描被R复位实测100Hz,VD366快100倍
+R     1.0, VD366            // VD_ExperimentDuration_Accum + 1(分钟)




// [已修复 v2.2] 删除 S5→S6 的 VD178 触发逻辑,统一由 FC40 双倒计时器写 VW2=7
 // [已修复 v2.2] 删除 S5→S6 的 VD178 触发逻辑,统一由 FC40 双倒计时器写 VW2=7




// 实验时长达标 - 转 S7 实验结束
       // 实验时长达标 - 转 S7 实验结束
// VD_ExperimentDuration_Accum >= VD_ExperimentTarget → 实验结束
 // VD_ExperimentDuration_Accum >= VD_ExperimentTarget → 实验结束
// 同时检查换水次数: VW400 >= VD414 (24h 换水目标次数)
 // 同时检查换水次数: VW400 >= VD414 (24h 换水目标次数)
LD     Always_On:SM0.0
LPS
AR>=   VD366, VD24           // 累计时长 >= 目标时长(min)
ITD    VW400, AC0            // 换水次数 INT → DINT 【v2.3.2迁移: 原VW306与手动命令位V306.0~V307.3重叠】
DTR    AC0, AC0              // → REAL
AR>=   AC0, VD414            // 【v2.2 新增】换水次数 >= 目标次数
R      T41, 1                // 停周期计时
R      T60, 1                // 停下缸满计时器
R      M10.7, 1              // 清预规划标志
MOVW   8, VW2                // →S7 (VW2=8)
LPP




// 注: v2.2 S5 不再调 FC40 预规划(三层纠偏已删除)
 // 注: v2.2 S5 不再调 FC40 预规划(三层纠偏已删除)
// 注: v2.2 S5 不再触发 VW2=1(上缸配液,改由 FC40 M16.1 触发下一轮 S1)
 // 注: v2.2 S5 不再触发 VW2=1(上缸配液,改由 FC40 M16.1 触发下一轮 S1)
// 注: v2.2 S5 不再调用 RhythmCorrection (FC40 改由 OB1 顶层调度,见 OB1 NET 6.5)
 // 注: v2.2 S5 不再调用 RhythmCorrection (FC40 改由 OB1 顶层调度,见 OB1 NET 6.5)
// 注: 周期阈值 VD186 在每周期 OB1 NET 6.5 调 FC40 时计算并刷新
 // 注: 周期阈值 VD186 在每周期 OB1 NET 6.5 调 FC40 时计算并刷新
// 注: HMI 手动停止命令由 FC2 统一处理(S1~S6 均响应),FC16 不再单独处理
 // 注: HMI 手动停止命令由 FC2 统一处理(S1~S6 均响应),FC16 不再单独处理
// 注: 断电恢复由 FC0 统一处理,VW2=6 (S5 无阀门动作) 时 FC0 保持 S5 并重算 VD_S5_Elapsed
 // 注: 断电恢复由 FC0 统一处理,VW2=6 (S5 无阀门动作) 时 FC0 保持 S5 并重算 VD_S5_Elapsed


// ============================================================
 // ============================================================
// 文件结束
                     // 文件结束
// ============================================================
 // ============================================================


END_SUBROUTINE_BLOCK

SUBROUTINE_BLOCK State_S6_Drain:SBR12
TITLE=// ============================================================
// // 文件: FC17_State_S6_Drain.stl
// // 功能: S6 下缸排水 (VW2=7)
// // Story: v2.2 流程重构 (替代 AQEX-6 状态机骨架 + AQEX-7 阀门诊断)
// // 说明: v2.2 S6 完成后状态转移按 VW418 分支:
// //       - VW418=3 (上缸已配完) + 结束条件满足 → S7
// //       - VW418=3 (上缸已配完) + 结束条件未满足 → S4 (VW2=5, 启动转移) + VW400+1 + M16.0 切
// //       - VW418≠3 (上缸未配完) → 保持等待,不报警
// //       后续下一轮 S1 由 FC40 (M16.1 触发条件) 在 FC15 S4 完成后切 M16.0 时启动
// // 【v10.4硬件变更】VW276=VD_Timeout_ValveC(VD54)×10、VW284=VD_Delay_ValveC_Verify(VD472)×10【2026-09-24由VD60迁来】,
// //       由本FC计算写入,供FC32(阀C诊断)作T56/T57/T58/T101的PT
// // ============================================================
BEGIN
Network 1
//  S6 首次进入动作 - 开阀C
//  [已修复 v2.2] 用 V62.0 缓存 EU 结果,避免 LPS/LPP 内 S/R 链栈空
LD     M10.7                 // S6 首次进入脉冲(FC16 NET 3 触发 M10.7 后)
EU
=      V62.0
LD     V62.0
EU                           // 开阀C
LD     V62.0
R      T42, 1
LD     SM0.0
TON    T42, 32767
LD     V62.0
MOVB   1, VB264
LD     V62.0
MOVB   0, VB265
LD     V62.0
MOVW   0, VW270
// 计算 VD_Timeout_ValveC(VD54)×10 转换值 // 计算 VD_Timeout_ValveC(VD54)×10 转换值
LD     V62.0
MOVR   VD54, VD328
*R     10.0, VD328
ROUND  VD328, AC0
MOVW   AC0, VW276
// 计算 VD_Delay_ValveC_Verify(VD472)×10 转换值【v10.4硬件变更新增】 // 计算 VD_Delay_ValveC_Verify(VD472)×10 转换值【v10.4硬件变更新增】
// 【2026-09-24迁移】原VD60废弃：VB60~VB63与v2.2修复的V60.x~V63.x EU缓存位区重叠, // 【2026-09-24迁移】原VD60废弃：VB60~VB63与v2.2修复的V60.x~V63.x EU缓存位区重叠,
//   每扫描周期被各FC的"= V6x.x"线圈重写, 浮点值闪变/变NaN(位型污染), 迁至VD472(全程序无占用) //   每扫描周期被各FC的"= V6x.x"线圈重写, 浮点值闪变/变NaN(位型污染), 迁至VD472(全程序无占用)
LD     V62.0
MOVR   VD472, VD328
*R     10.0, VD328
ROUND  VD328, AC0
MOVW   AC0, VW284
// 调用阀C诊断                    // 调用阀C诊断
LD     SM0.0
CALL ValveC_Diag
// 检查阀C诊断结果                  // 检查阀C诊断结果
// [已修复 v2.2] 用 V62.1 缓存诊断完成条件,避免 LPS/LPP+NOT 配合下的 S/R 链栈空 // [已修复 v2.2] 用 V62.1 缓存诊断完成条件,避免 LPS/LPP+NOT 配合下的 S/R 链栈空
LD     SM0.0
=      V62.0                 // 阀C诊断正常完成(VB270=1)
=      V62.1
LDN    V62.1
LD     V62.0                 // 未完成 → 跳过
// 【v2.3修复】先读T42当前值再复位(R在前读到的恒为0) // 【v2.3修复】先读T42当前值再复位(R在前读到的恒为0)
LD     V62.1
MOVW   T42, AC0
S      CPU_输出4:Q0.4, 1       // → DINT
DTR    VD444, VD444
LD     V62.0                 // 【v2.3.6】100ms时基→秒                // → REAL(原值秒)
LD     V62.1
R      T42, 1                // VD116 = S6 实测秒(后续轮次用)
LD     V62.1
LD     Always_On:SM0.0       // 停S6计时(读后复位)
LD     V62.1
TON    T42, 32767            // 【v2.3修复】排水完成→下缸=空
                                   // (原无任何FC在S6完成时清V1.7, 下一轮S4的"AN V1.7" // (原无任何FC在S6完成时清V1.7, 下一轮S4的"AN V1.7"
                                   //  永不满足, 换水循环在第二轮起卡死) //  永不满足, 换水循环在第二轮起卡死)
LBL    10
// 排水完成 → 状态转移 (v2.2 按 VW418 分支) // 排水完成 → 状态转移 (v2.2 按 VW418 分支)
//
// 情况 1: 上缸已配完 (VW418=3) + 结束条件满足 → S7 // 情况 1: 上缸已配完 (VW418=3) + 结束条件满足 → S7
LD     SM0.0
LD     V62.0                 // 上缸已配完
MOVB   1, VB264              // 无报警(FC3 管理)
LPS
LD     V62.0                 // 实验时长累计 >= 目标(min)
LPP
LPS
MOVB   0, VB265              // 换水次数 INT → DINT 【v2.3.2迁移: 原VW306与手动命令位V306.0~V307.3重叠】
LD     V62.0                 // → REAL
MOVW   0, VW270              // 换水次数 >= 目标
LPP
LD     V62.0                 // 两个结束条件同时满足
NOT
MOVR   VD54, VD328           // 不满足 → 检查情况 2
*R     10.0, VD328           // → S7
ROUND  VD328, AC0            // 跳到末尾
LBL    11
// 情况 2: 上缸已配完 (VW418=3) + 结束条件未满足 → S4 + 计数 + 切计时器 // 情况 2: 上缸已配完 (VW418=3) + 结束条件未满足 → S4 + 计数 + 切计时器
LD     SM0.0
MOVW   AC0, VW276            // 上缸已配完
LD     V62.0                 // 无报警
NOT
MOVR   VD472, VD328          // 上缸未配完 → 情况 3
*R     10.0, VD328           // → S4 (转移)
ROUND  VD328, AC0            // 换水计数 +1 【v2.3.2迁移: 原VW306与手动命令位V306.0~V307.3重叠】
LD     M16.0
NOT
MOVW   AC0, VW284            // 切双倒计时器标记
JMP    13
LBL    12
// 情况 3: 上缸未配完 (VW418≠3) → 保持等待,不报警 // 情况 3: 上缸未配完 (VW418≠3) → 保持等待,不报警
// 无动作,等上缸配完自然进 S4           // 无动作,等上缸配完自然进 S4
// 注: 此时 V1.7=0(已排空)但上缸未配完,系统空转等待 // 注: 此时 V1.7=0(已排空)但上缸未配完,系统空转等待
//      不会触发 24h 换水次数超时报警(那是 FC40 VD248/VD252 >= T_cycle 才报) //      不会触发 24h 换水次数超时报警(那是 FC40 VD248/VD252 >= T_cycle 才报)
LBL    13
// 注: 【v10.4硬件变更】FC32已改为「液位低位+VD_Delay_ValveC_Verify延时验证」判定排水完成 // 注: 【v10.4硬件变更】FC32已改为「液位低位+VD_Delay_ValveC_Verify延时验证」判定排水完成
//      开关到位、超时保护仍由 FC32 统一处理 //      开关到位、超时保护仍由 FC32 统一处理
// 注: VD_S6_Rolling 滚动平均算法由 FC17 直接覆盖(简单实现) // 注: VD_S6_Rolling 滚动平均算法由 FC17 直接覆盖(简单实现)
// 注: 断电恢复由 FC0 统一处理,VW2=7 (S6 阀C动作中断) 时 FC0 转 S_ERROR // 注: 断电恢复由 FC0 统一处理,VW2=7 (S6 阀C动作中断) 时 FC0 转 S_ERROR
// 注: 【v2.2】原"实验未结束 → S5,已结束 → S7"二元判断改为三元判断(增加上缸配完分支) // 注: 【v2.2】原"实验未结束 → S5,已结束 → S7"二元判断改为三元判断(增加上缸配完分支)
// ============================================================ // ============================================================
// 文件结束                      // 文件结束
// ============================================================

 // ============================================================
LD     Always_On:SM0.0
CALL   ValveC_Diag:SBR18
LD     Always_On:SM0.0
AB=    VB270, 1
=      V62.1
LDN    V62.1
JMP    10
LD     V62.1
MOVW   T42, AC0
ITD    AC0, VD444
DTR    VD444, VD444
/R     10.0, VD444
LD     V62.1
MOVR   VD444, VD116
LD     V62.1
R      T42, 1
LD     V62.1
R      V1.7, 1
LBL    10
LD     Always_On:SM0.0
AW=    VW418, 3
AW=    VW6, 0
LPS
AR>=   VD366, VD24
LPP
LPS
ITD    VW400, AC0
DTR    AC0, AC0
AR>=   AC0, VD414
LPP
ALD
NOT
JMP    11
MOVW   8, VW2
JMP    13
LBL    11
LD     Always_On:SM0.0
AW=    VW418, 3
AW=    VW6, 0
NOT
JMP    12
MOVW   5, VW2
INCW   VW400
LD     M16.0
NOT
=      M16.0
JMP    13
LBL    12
LBL    13
END_SUBROUTINE_BLOCK

SUBROUTINE_BLOCK State_S7_End:SBR13
TITLE=// ============================================================
// // 文件: FC18_State_S7_End.stl
// // 功能: S7实验结束 (VW2=8)
// // Story: AQEX-6 状态机骨架
// // 说明: 实验完成，状态锁定，提示人工按系统复位后回S0
// // ★ v10重大变更: S7彻底屏蔽V0.0(CMD_Start),只响应I0.3(系统复位按钮)
// //   原实现V0.0↑→回S0,但FC10启动还需再按一次,两次按钮才能启动
// //   且V0.0在S7语义不干净(按钮名叫"启动"实际是"清计数器回S0")
// //   改后:S7唯一出口是物理I0.3系统复位按钮,回S0后V0.0正常工作
// //   实验结束提示由HMI侧用 VW2=8 条件弹窗（原V301.7为预留扩展位,已废弃）
// // ============================================================
// 
BEGIN
Network 1
//  S7进入动作 - 安全停机
LD     Always_On:SM0.0
// 复位Q0.0~Q0.6(泵/阀),Q0.7/Q8.0报警声光由FC3统一管理,避免与FC3双写导致闪亮
 // 复位Q0.0~Q0.6(泵/阀),Q0.7/Q8.0报警声光由FC3统一管理,避免与FC3双写导致闪亮
// 【v10.4硬件变更】Q0.6(下缸NC阀)已去除,保留未使用;R Q0.0,7清零无害
 // 【v10.4硬件变更】Q0.6(下缸NC阀)已去除,保留未使用;R Q0.0,7清零无害
R      CPU_输出0:Q0.0, 7       // 泵停、阀A/B/C关,保留Q0.7
// 停止实验时长累加(VD_ExperimentDuration_Accum锁定最终值)
 // 停止实验时长累加(VD_ExperimentDuration_Accum锁定最终值)
R      T47, 1                // 停1分钟基准计时
// 置实验结束标志(供S6判断是否走最终排水→S7路径)
 // 置实验结束标志(供S6判断是否走最终排水→S7路径)
S      M10.6, 1




// S7唯一出口 — 物理系统复位按钮I0.3（原 NETWORK 3，NETWORK 2 已废弃）
 // S7唯一出口 — 物理系统复位按钮I0.3（原 NETWORK 3，NETWORK 2 已废弃）
// 注：原 NETWORK 2 每周期 S V301.7 提示位已废弃，改为 HMI 侧用 VW2=8 条件弹窗
 // 注：原 NETWORK 2 每周期 S V301.7 提示位已废弃，改为 HMI 侧用 VW2=8 条件弹窗
// v10重写: S7彻底屏蔽V0.0(CMD_Start),只响应I0.3(系统复位按钮)
 // v10重写: S7彻底屏蔽V0.0(CMD_Start),只响应I0.3(系统复位按钮)
// 原实现: V0.0↑→回S0 (已删除,改由I0.3负责)
 // 原实现: V0.0↑→回S0 (已删除,改由I0.3负责)
// 复位条件(全部满足):
              // 复位条件(全部满足):
//   I1.1=OFF 急停已释放(和FC19/S_ERROR复位保持一致)
 //   I1.1=OFF 急停已释放(和FC19/S_ERROR复位保持一致)
//   I0.3上升沿 系统复位按钮按下(就地面板物理按钮,非HMI软命令)
 //   I0.3上升沿 系统复位按钮按下(就地面板物理按钮,非HMI软命令)
// 为什么S7用I0.3不用V0.0:
        // 为什么S7用I0.3不用V0.0:
//   - V0.0语义是"启动实验",在S7里用它回S0是双重语义,不干净
 //   - V0.0语义是"启动实验",在S7里用它回S0是双重语义,不干净
//   - 改后V0.0只在S0有效,按钮语义单一
  //   - 改后V0.0只在S0有效,按钮语义单一
//   - 物理复位按钮比HMI软命令更安全(实验结束后强制人工确认)
 //   - 物理复位按钮比HMI软命令更安全(实验结束后强制人工确认)
LDN    CPU_输入9:I1.1          // 急停已释放(常闭触点恢复ON=正常)
A      CPU_输入3:I0.3          // 系统复位按钮按下
EU                           // 上升沿(按下瞬间触发一次)
// 清实验结束标志
                  // 清实验结束标志
R      M10.6, 1
// 清握手位(由S0重新管理)
            // 清握手位(由S0重新管理)
R      V1.0, 1
// 清零本次实验累计值,准备新一轮
          // 清零本次实验累计值,准备新一轮
MOVR   0.0, VD406            // 清累计流量 (原VD364,2026-09-29迁移:与VD366重叠2字节;VD402槽被VW402(T38_PT)占)
MOVR   0.0, VD440            // 清累计加药量
MOVR   0.0, VD372            // 清S3剩余待加药量
// 状态回S0,后续由FC10接管
          // 状态回S0,后续由FC10接管
MOVW   0, VW2




// ============================================================
 // ============================================================
// 文件结束
                     // 文件结束
// ============================================================
 // ============================================================


END_SUBROUTINE_BLOCK

SUBROUTINE_BLOCK State_Error:SBR14
TITLE=// ============================================================
// // 文件: FC19_State_Error.stl
// // 功能: S_ERROR故障锁定 (VW2=99)
// // Story: AQEX-6 状态机骨架 + AQEX-9 急停双通道+安全继电器反馈(详细实现) + AQEX-10 编址修正(V0.5→V0.7)
// // 说明: 急停或最高级报警触发后的故障锁定,强制输出安全状态
// //       继电器故障(V300.5)禁止复位,必须HMI高权限确认(V0.7)+I1.2正常后清除
// // 急停解除(I1.1=OFF,NO 触点释放)+系统复位按钮(I0.3)→回S0  v1.3 改 NO 接法
// // ============================================================
// 
// // 符号说明:
// // I1.1  : DI_EStop           急停反馈(常开 NO,OFF=正常,ON=急停触发)  v1.3 改为接 NO 触点
// // I1.2  : DI_SafetyRelay_FB  安全继电器辅助反馈(ON=动力回路已断开确认)
// // I0.3  : DI_Btn_SystemReset 系统复位按钮(无源常开点动)
// // V0.7  : CMD_SafetyRelayAck HMI高权限确认继电器故障已检修(需二次确认/高权限)
// // V300.4: M_EStop_Latch      急停触发锁存(漫溢级)
// // V300.5: M_Alarm_SafetyRelay 安全继电器故障(最高级)
// // V1.6  : M_TankA_State      上缸状态(0=空,1=满)
// // V1.7  : M_TankB_State      下缸状态(0=空,1=满)
// // VW2   : 状态机状态(FC19写0回S0)
// // VW6   : 报警码
// 
// 
BEGIN
Network 1
//  故障态输出强制安全(与FC2 NETWORK3双保险)
//  S_ERROR态双保险:即使FC2未执行,QB0也强制安全
LD     Always_On:SM0.0
MOVB   0, QB0                // 潜水泵停/阀关/上缸NC阀失电(关闭=安全;Q0.6已去除,保留未使用)
S      CPU_输出7:Q0.7, 1       // 报警声音(FC3管理消音)
// Q8.0灯光由FC3按报警优先级管理(急停/继电器故障=常亮)
 // Q8.0灯光由FC3按报警优先级管理(急停/继电器故障=常亮)




// 继电器故障禁止复位检测
              // 继电器故障禁止复位检测
// 9.4: 继电器故障不允许任何自动恢复,必须人工检修
 // 9.4: 继电器故障不允许任何自动恢复,必须人工检修
// V300.5=1时,即使I1.1恢复+I0.3按下,也不允许回S0
 // V300.5=1时,即使I1.1恢复+I0.3按下,也不允许回S0
LD     V300.5                // 继电器故障=1
JMP    1                     // 跳过系统复位,转NETWORK4检查HMI确认
// V300.5=0(无继电器故障) → 继续NETWORK3系统复位
 // V300.5=0(无继电器故障) → 继续NETWORK3系统复位




// 急停解除+系统复位按钮 → 回S0
        // 急停解除+系统复位按钮 → 回S0
// 复位条件(全部满足):
              // 复位条件(全部满足):
//   I1.1=OFF(急停按钮已释放,NO 触点恢复)
 //   I1.1=OFF(急停按钮已释放,NO 触点恢复)
//   I0.3上升沿(系统复位按钮按下)
      //   I0.3上升沿(系统复位按钮按下)
//   V300.5=0(NETWORK2已确认无继电器故障)
 //   V300.5=0(NETWORK2已确认无继电器故障)
LDN    CPU_输入9:I1.1          // 急停已释放(常开 NO 触点恢复 OFF)  v1.3 改 NO 接法
A      CPU_输入3:I0.3          // 系统复位按钮按下
EU                           // 上升沿(按下瞬间)
=      V61.0                 // [已修复 v2.2] 缓存 EU 结果,避免后续 R 指令链栈空
// 清急停锁存
                    // 清急停锁存
LD     V61.0
R      V300.4, 1             // M_EStop_Latch=0
// 清漫溢级报警(这些锁存位需系统复位清除)
     // 清漫溢级报警(这些锁存位需系统复位清除)
// 【v10.4硬件变更】V300.3已废弃为保留位(下缸NC阀Q0.6去除),仍一并清零无害
 // 【v10.4硬件变更】V300.3已废弃为保留位(下缸NC阀Q0.6去除),仍一并清零无害
LD     V61.0
R      V300.0, 4             // V300.0~V300.3=0
// 【2026-09-29修复】系统复位同时清一般故障级报警位V301~V303
 // 【2026-09-29修复】系统复位同时清一般故障级报警位V301~V303
// 原因: 阀A开到位超时(V301.4)等报警的自动复位条件是"物理条件消失"(如I8.0=ON),
 // 原因: 阀A开到位超时(V301.4)等报警的自动复位条件是"物理条件消失"(如I8.0=ON),
//   但阀关闭的待机态与故障态同为I8.0=OFF,条件复位永远等不到; 而FC10启动门槛要求VW6=0,
 //   但阀关闭的待机态与故障态同为I8.0=OFF,条件复位永远等不到; 而FC10启动门槛要求VW6=0,
//   形成死锁(报警消不掉+无法重启)。系统复位=系统级人工确认;
 //   形成死锁(报警消不掉+无法重启)。系统复位=系统级人工确认;
//   复位后故障若仍存在会被各FC重新置位重新报警,不会丢失故障。
 //   复位后故障若仍存在会被各FC重新置位重新报警,不会丢失故障。
// 注: V303.6(周期超时)在此清位安全——VD248/252双计时器已在下方同批清零,
 // 注: V303.6(周期超时)在此清位安全——VD248/252双计时器已在下方同批清零,
//   不会同扫描被FC40 NET6重报(问题#6死锁对策已具备)
 //   不会同扫描被FC40 NET6重报(问题#6死锁对策已具备)
LD     V61.0
R      V301.0, 8             // 阀A类全部(V301.0~V301.7)
LD     V61.0
R      V302.0, 8             // 阀B/C类全部(V302.0~V302.7)
LD     V61.0
R      V303.0, 8             // 阀C/注射泵/RTC/周期超时全部(V303.0~V303.7)
// 强制上下缸状态置空(9.3:复位后上下缸状态强制置"空")
 // 强制上下缸状态置空(9.3:复位后上下缸状态强制置"空")
LD     V61.0
R      V1.6, 1               // 上缸=空
LD     V61.0
R      V1.7, 1               // 下缸=空
// ★ 2026-09-11 新增: 清阀门诊断子状态和计时器
 // ★ 2026-09-11 新增: 清阀门诊断子状态和计时器
// 与OB1停止命令同根因: FC11/FC15/FC17的AW=VW2xx,0前置条件
 // 与OB1停止命令同根因: FC11/FC15/FC17的AW=VW2xx,0前置条件
LD     V61.0
FILL   0, VW260, 8           // 清 VB260~VB275 (阀A/B/C 诊断)
LD     V61.0
R      T50, 6                // 清 T50~T55 (阀A/B 诊断计时器)
// 转S0初始化(9.3:回到S0重新开始,不支持从中断点继续)
 // 转S0初始化(9.3:回到S0重新开始,不支持从中断点继续)
LD     V61.0
MOVW   0, VW2                // VW2=0(S0)
// 清报警码
                     // 清报警码
LD     V61.0
MOVW   0, VW6
// 清启动命令残留,防止复位后MCGS残留V0.0=1导致立即重启动
 // 清启动命令残留,防止复位后MCGS残留V0.0=1导致立即重启动
LD     V61.0
R      V0.0, 1
// 【2026-09-29新增】清S1首次进入标志(与VW418清零配套,防止复位后S1门控残留)
 // 【2026-09-29新增】清S1首次进入标志(与VW418清零配套,防止复位后S1门控残留)
LD     V61.0
R      M10.2, 1
// 停报警声音(灯光由FC3按确认流程管理)
     // 停报警声音(灯光由FC3按确认流程管理)
LD     V61.0
R      CPU_输出7:Q0.7, 1
// ★ 2026-09-24 新增: 清上缸子流程状态 + 双倒计时器标志 + 定时器
 // ★ 2026-09-24 新增: 清上缸子流程状态 + 双倒计时器标志 + 定时器
//   与OB1停止命令块/SBR26同款清理, 修复"系统复位后VW418残留→上缸跳过S1自启动"
 //   与OB1停止命令块/SBR26同款清理, 修复"系统复位后VW418残留→上缸跳过S1自启动"
LD     V61.0
MOVW   0, VW418              // 上缸配液子流程状态清零
LD     V61.0
MOVW   0, VW400              // 换水计数清零
LD     V61.0
R      M16.0, 4              // M16.0~M16.3 连续清零(双倒计时器标志+S1/S2首次进入门控)
LD     V61.0
R      T38, 1                // 清 S2 搅拌定时器
LD     V61.0
R      T63, 1                // 清 1s 脉冲定时器
LD     V61.0
R      T49, 1                // 清 S4 转移计时器
LD     V61.0
MOVR   0.0, VD248            // 清 TimerA_Elapsed
LD     V61.0
MOVR   0.0, VD252            // 清 TimerB_Elapsed
LD     V61.0
MOVR   0.0, VD256            // 清 TimerA 显示值
LD     V61.0
MOVR   0.0, VD244            // 清 TimerB 显示值
JMP    2                     // 复位完成,结束




